// TwinCAT 3 PLC project RACBaseObjects
// Title: Base Objects Library
// Company: JABIL RAC LATAM
// Author: RAC Team
// ProjectVersion: 24.12.1
// Description: Base library for base devices and machines in RAC LATAM
// ProgramVersion: 3.1.4024.0
// libraries:
//   Tc2_MC2, * (Beckhoff Automation GmbH)
//   Tc2_Standard, * (Beckhoff Automation GmbH)
//   Tc2_System, * (Beckhoff Automation GmbH)
//   Tc3_Module, * (Beckhoff Automation GmbH)
// project tree:
//   DUTs/ ST_Nest.TcDUT, ST_RAC_EIP.TcDUT
//   GVLs/ Constants.TcGVL, GVL_Rails.TcGVL
//   / PlcTask.TcTTO
//   POUs/00_Interfaces/Device/ FB_Device.TcPOU, ST_Alarm.TcDUT
//   POUs/00_Interfaces/Machine/ FB_Machine.TcPOU
//   POUs/00_Interfaces/Stations/ EN_StationStatus.TcDUT, FB_Station.TcPOU
//   POUs/01-DevicesFB/Bimanual/ FB_Bimanual.TcPOU (not stored)
//   POUs/01-DevicesFB/BowlFeeder/ ST_BowlFeeder.TcDUT
//   POUs/01-DevicesFB/Conveyor/ FB_Conveyor.TcPOU
//   POUs/01-DevicesFB/Cylinder/ FB_Cylinder.TcPOU
//   POUs/01-DevicesFB/LightTower/ FB_LightTower.TcPOU
//   POUs/01-DevicesFB/Motor/ EN_MotionType.TcDUT, FB_Motor.TcPOU
//   POUs/01-DevicesFB/RejectCar/ FB_RejectCart.TcPOU
//   POUs/01-DevicesFB/Robot/ EN_RobotMessaging.TcDUT, FB_Robot.TcPOU, ST_RobotIO.TcDUT
//   POUs/01-DevicesFB/Scanner/ FB_Scanner.TcPOU
//   POUs/01-DevicesFB/TrayFeeder/ EN_TrayFeederMessaging.TcDUT, FB_TrayFeeder.TcPOU, ST_TrayFeederIO.TcDUT
//   POUs/01-DevicesFB/Vaccum/ FB_Vacuum.TcPOU
// real-time tasks:
//   TASK PlcTask: cycle T#10ms, priority 20, ADS port 350

CONFIGURATION RACBaseObjects
    RESOURCE PLC ON TwinCAT3
        TASK PlcTask(INTERVAL := T#10ms, PRIORITY := 20);
    END_RESOURCE
END_CONFIGURATION

// ---- DUTs/ST_Nest.TcDUT
TYPE ST_Nest :
	STRUCT
		railSerial				: STRING;
		controllerSerial		: STRING;
		batterySerial			: STRING;
		nestID					: USINT;
		conveyorPosition		: USINT;
		okToProcess				: BOOL				:= FALSE;
		failureMode				: STRING			:= 'N/A';
		endcapAssembled			: BOOL 				:= FALSE;
		controllerAssembled		: BOOL				:= FALSE;	
	END_STRUCT
END_TYPE

// ---- DUTs/ST_RAC_EIP.TcDUT
TYPE ST_RAC_EIP :
STRUCT
	byteArray 		: ARRAY [0..39] OF BYTE;
END_STRUCT
END_TYPE

// ---- POUs/00_Interfaces/Device/ST_Alarm.TcDUT
TYPE ST_Alarm :
STRUCT
	sCode							: STRING;
	bIsActive						: BOOL;
	bWrittenOnGeneralAlarm			: BOOL;
END_STRUCT
END_TYPE

// ---- POUs/00_Interfaces/Stations/EN_StationStatus.TcDUT
{attribute 'qualified_only'}
{attribute 'strict'}
{attribute 'to_string'}
TYPE EN_StationStatus :
(
	estopped			:=0,
	stopped				:=1,
	maintenance			:=2,
	initializing		:=3,
	idle				:=4,
	running				:=5
	);
END_TYPE

// ---- POUs/01-DevicesFB/BowlFeeder/ST_BowlFeeder.TcDUT
TYPE ST_BowlFeeder :
	STRUCT
		bOut_Vibrate			AT%Q*	: BOOL;
		bOut_BlowAlign			AT%Q*	: BOOL;
		bIn_NoMaterial			AT%I*	: BOOL;
		bIn_LowLevelMaterial	AT%I*	: BOOL;
		bIn_UnitInPosition		AT%I*	: BOOL;
	END_STRUCT
END_TYPE

// ---- POUs/01-DevicesFB/Motor/EN_MotionType.TcDUT
{attribute 'qualified_only'}
{attribute 'strict'}
{attribute 'to_string'}
TYPE EN_MotionType :
(
	idle 			:= 0,
	stop 			:= 1,
	home 			:= 2,
	jogPos 			:= 3,
	jogNeg 			:= 4,
	absolute 		:= 5,
	relative 		:= 6
);
END_TYPE

// ---- POUs/01-DevicesFB/Robot/EN_RobotMessaging.TcDUT
{attribute 'qualified_only'}
{attribute 'strict'}
{attribute 'to_string'}
TYPE EN_RobotMessaging :
(
	clearedCmd 					:=10000,
	ok							:=10001,
	retry						:=10002,
	skip						:=10003,
	retriesExceeded				:=10004,
	
	initStart					:=0,
	waitInitPermissive			:=10,
	turnMotorsOFF				:=20,
	waitRobotInAuto				:=30,
	resetEStop					:=40,
	PPToMain					:=50,
	turnMotorsON				:=60,
	startTaskExecuion			:=70,
	waitInitFinihsed			:=80,
	waitRetrievalPerm			:=210,
	stopTaskExecution			:=310,
	initEndMotorsOFF			:=320,
	initFinished				:=999,
	
	autoStarts					,
	waitingPickPerm				,
	pickingGood					,
	pickingNG					,
	waitingPieceStatus			,
	waitingPlacePerm			,
	placing						,
	placeFinished				,
	waitingRejectPerm			,
	rejecting					,
	rejectFinished				,
	autoCycleFinished			:=1999,
	
	manualRetrieval				,
	manualHomming				,
	manualPick					,
	manualCycPickTeach			,
	manualPlace					,
	manualCycPlaceTeach			,
	manualReject				,
	manualCycRejectTeach		
)DINT := clearedCmd;
END_TYPE

// ---- POUs/01-DevicesFB/Robot/ST_RobotIO.TcDUT
TYPE ST_RobotIO :
STRUCT
	uiin_ConnectionStatus					AT %I*		:UINT;
	eipInputs								AT %I*		:ST_RAC_EIP;
	eipOutputs								AT %Q*		:ST_RAC_EIP;
	
	diin_Sequencer		 					:DINT;
	diout_SequenceCmd						:DINT;
	rout_XCompensation						:REAL;
	rout_ZCompensation						:REAL;
	
	bin_EStop	 							:BOOL;
	bin_PPMoved	 							:BOOL;
	bin_MotorsOFF	 						:BOOL;
	bin_MotorsON	 						:BOOL;
	bin_SystemInputBusy	 					:BOOL;
	bin_RunchainOK	 						:BOOL;
	bin_AutoON	 							:BOOL;
	bin_MainTaskExecuting	 				:BOOL;
	bin_SMBBatery	 						:BOOL;
	bin_RobotNotMoving						:BOOL;
	
	bout_ResetEStop							:BOOL;
	bout_PPToMain							:BOOL;
	bout_MotorsOFF							:BOOL;
	bout_MotorsON							:BOOL;
	bout_Start								:BOOL;
	bout_Stop								:BOOL;
	
	bin_almRetCyl01							:BOOL;
	bin_almExtCyl01							:BOOL;
	bin_almBothSnsrCyl01					:BOOL;
	bin_almRetCyl02							:BOOL;
	bin_almExtCyl02							:BOOL;
	bin_almBothSnsrCyl02					:BOOL;
	bin_almRetCyl03							:BOOL;
	bin_almExtCyl03							:BOOL;
	bin_almBothSnsrCyl03					:BOOL;
END_STRUCT
END_TYPE

// ---- POUs/01-DevicesFB/TrayFeeder/EN_TrayFeederMessaging.TcDUT
{attribute 'qualified_only'}
{attribute 'strict'}
{attribute 'to_string'}
TYPE EN_TrayFeederMessaging :
(
	waitInitStart			:=0,
	initFinished			:=999,
	
	autoStart				:=1000,
	readyToScan				:=1400,
	scanning				:=1410,
	scanFinished			:=1490,
	readyToPick				:=1500,
	picking					:=1510,
	pickFinished			:=1590,
	autoProcessFinished		:=1999
)DINT := waitInitStart;
END_TYPE

// ---- POUs/01-DevicesFB/TrayFeeder/ST_TrayFeederIO.TcDUT
TYPE ST_TrayFeederIO :
STRUCT
	uiin_ConnectionStatus					AT %I*		:UINT;
	eipInputs								AT %I*		:ST_RAC_EIP;
	eipOutputs								AT %Q*		:ST_RAC_EIP;
	
	diin_StationStatus						:DINT;
	diin_Sequencer		 					:DINT;
	diout_SequenceCmd						:DINT;
	
	bin_ServosFailure						:BOOL;
	bin_initFinished						:BOOL;
	bin_AutoOn								:BOOL;
	bin_eStop								:BOOL;
	
	bout_Reset								:BOOL;
	bout_Start								:BOOL;
	bout_Stop								:BOOL;
	bout_Init_startPermissive				:BOOL;
	
	bout_readyToScan						:BOOL;
	bout_readyToPick						:BOOL;
	bin_SafetyBoxPlace_OutOfZone	 		:BOOL;
	bout_SafetyBoxPlace_Permissive 			:BOOL;
	
	bin_inScanningPosition					:BOOL;
	bout_scannninPieceIsOK					:BOOL;
	bout_scannninPieceIsNG					:BOOL;
	
	bin_delivery_trayReady					:BOOL;
	bout_delivery_trayChangeRequest			:BOOL;
END_STRUCT
END_TYPE

// ---- GVLs/Constants.TcGVL
{attribute 'qualified_only'}
VAR_GLOBAL CONSTANT
	
	Total_Nest						: USINT		:= 155;
	
	LoadPos							: USINT		:= 1;
	NestScanPos						: USINT		:= 2;
	EndcapAsmPos					: USINT		:= 3;
	ControllerScanPos				: USINT		:= 4;	
	BatteryConnectPos		 		: USINT		:= 5;
	ControllerAsmPos				: USINT		:= 6;
	DisplayScanPos		 			: USINT		:= 18;	
	BatteryDisconnectPos			: USINT		:= 20;
	TappingPos						: USINT		:= 23;
	
//	St01_LoadPos					: USINT		:= 1; // From quiles branch 
//	St01_EndcapAsmPos				: USINT		:= 3;
//	St01_ControllerAsmPos				: USINT		:= 4;
//	St01_BatteryAsmPos				: USINT		:= 5;
//	St01_UnloadPos					: USINT		:= 9;
						
END_VAR

// ---- GVLs/GVL_Rails.TcGVL
{attribute 'qualified_only'}
VAR_GLOBAL
		Nests	: ARRAY[1..Constants.Total_Nest] OF ST_Nest;
	
END_VAR

// ---- POUs/00_Interfaces/Device/FB_Device.TcPOU
FUNCTION_BLOCK  FB_Device
VAR_INPUT
	// Status of Master station
	diStationState 						: EN_StationStatus;
	
	// Device Identification Number
	sDeviceID							: STRING;
	
	// Stop executions
	bStopExecution						: BOOL;
	
	// Station Alarm Reset
	bAlarmReset							: BOOL;
END_VAR
VAR_OUTPUT
	// Display current active alarms in device, in a CVS file concatenating type string
	sAlarm								: STRING;
END_VAR
VAR RETAIN
	// Var to set timeout value in each step
	tmStepTimeout						: TIME		:=T#1S;
	
	// General timeout TON
	ton_StepTimeout						: TON;
	// Pulse ton
	ton_pulse							: TON;
END_VAR

METHOD AlarmCodesHandling : STRING
VAR_INPUT
	// Concatenated codes string
	sConcatCodes						:	STRING;
	// Code for add or delete
	sCode								:	STRING;
	// Device ID for add to alarm code
	sIDToAdd							:	STRING;
	// If alarm is active: TRUE
	bActive								:	BOOL;
END_VAR
VAR
	// Code with ID and separator added
	sProcessedCode						:	STRING;
	// Position where code was found
	iPosWhereFindCode					:	INT;
	// Length of code seeked
	iLengthOfCode						:	INT;
END_VAR
//	Add device ID, separator, seek code in concatenated codes string obtan position in the string and lentgh of seeked code
	sProcessedCode:= CONCAT(STR1:=sCode,STR2:=sIDToAdd);
	sProcessedCode:= CONCAT(STR1:=sProcessedCode,STR2:=',');
	iPosWhereFindCode:= FIND(STR1:=sConcatCodes,STR2:=sProcessedCode);
	iLengthOfCode:= LEN(STR:=sProcessedCode);

//	If code was not found add alarm is active add it to concatenated codes string
	IF (iPosWhereFindCode=0) AND (bActive) THEN
		AlarmCodesHandling:= CONCAT(STR1:=sConcatCodes,STR2:=sProcessedCode);
//	If code was found add alarm is not active delete it from concatenated codes string
	ELSIF (iPosWhereFindCode<>0) AND (NOT bActive) THEN
		AlarmCodesHandling:= DELETE(STR:=sConcatCodes,LEN:=iLengthOfCode,POS:=iPosWhereFindCode);
//	Default case return input value
	ELSE
		AlarmCodesHandling:= sConcatCodes;
	END_IF
END_METHOD

END_FUNCTION_BLOCK

// ---- POUs/00_Interfaces/Machine/FB_Machine.TcPOU
FUNCTION_BLOCK ABSTRACT FB_Machine EXTENDS FB_Device
VAR_INPUT
	// Init start permissive
	bInit_StartPermissive				: BOOL;
END_VAR
VAR_OUTPUT
	// Init finished
	bInit_Finished						: BOOL;
END_VAR
VAR RETAIN
	// Sequencer
	diActualSeqStep						: DINT;
	
	// Var to follow sequencer and evaluate timeout	
	diLastActiveStep					: DINT;
END_VAR

METHOD ABSTRACT Alarm
END_METHOD

METHOD ABSTRACT Auto
END_METHOD

METHOD ABSTRACT Init
END_METHOD

METHOD ABSTRACT IO
END_METHOD

METHOD MachineMain
//	Enable Setting Alarm Routine Execution
	THIS^.IO();

//	Machine state control

CASE diStationState OF
	EN_StationStatus.stopped,
	EN_StationStatus.estopped:			//Enables Stop Routine Execution
		THIS^.Stop();
	EN_StationStatus.initializing:		//Enables Init Routine Execution
		THIS^.Init();
	EN_StationStatus.idle:				//Enables Pause Routine
		THIS^.Pause();
	EN_StationStatus.running:			//Enables Auto Routine Execution
		THIS^.Auto();
	EN_StationStatus.maintenance:		//Enables Manual Routine Execution
		THIS^.Manual();
END_CASE

//	Enable Setting Alarm Routine Execution
	THIS^.Alarm();
END_METHOD

METHOD ABSTRACT Manual
END_METHOD

METHOD ABSTRACT Pause
END_METHOD

METHOD ABSTRACT Stop
END_METHOD

END_FUNCTION_BLOCK

// ---- POUs/00_Interfaces/Stations/FB_Station.TcPOU
FUNCTION_BLOCK FB_Station
VAR_INPUT
	// Whole Station Init finished
	bInitFinished						: BOOL;
	
	// All E-Stop buttons
	EmergencyStop 						: BOOL;
	// From safety project
	SafetyReady 						: BOOL;
	// All door sensors
	Interlock 							: BOOL;
END_VAR
VAR_OUTPUT
	// Station Actual Status 
	diStationState 						: EN_StationStatus;
	
	// Stop executions
	bStop								: BOOL;
	
	// Reset Alarms
	 bAlarmReset						: BOOL;
END_VAR
VAR
	bStopButton 			AT %I* 		: BOOL;
	bStartButton 			AT %I* 		: BOOL;
	bResetButton			AT %I* 		: BOOL;

	bStopInterface 						: BOOL;
	bPauseInterface 					: BOOL;
	bInitStartInterface					: BOOL;
	bAutoStartInterface 				: BOOL;
	bResetInterface						: BOOL;
	OpUser 								: BOOL;

	AutoModeSelector 		AT %I* 		: BOOL;
	PressureSwitch 			AT %I* 		: BOOL;
	
	// Delay for stoppping machine with button 
	ton_stopMachineDelay 				: TON;
	
	// Delay for starts machine with button
	ton_startInitStartButtonDelay 		: TON;
END_VAR

StatusControl();
Alarm();

METHOD Alarm
VAR_INPUT
END_VAR
END_METHOD

METHOD StatusControl
VAR_INPUT
END_VAR

VAR
	// Safe operation condition in any mode
	bSafeOperationCondition			: BOOL;
	
	// Condtion for any Auto operation mode
	bAutoAvailable					: BOOL;
	
	// Condition for Maintenance operation mode
	bManualAvailable				: BOOL;
END_VAR
//	Condition for operate machine safely in any mode
	bSafeOperationCondition					:=	SafetyReady AND Interlock AND PressureSwitch;

//	Condition for operation in Auto Mode
	bAutoAvailable							:=	bSafeOperationCondition AND AutoModeSelector;

//	Condition for operation in Maintenance Mode
	bManualAvailable						:=	bSafeOperationCondition AND OpUser AND (NOT AutoModeSelector);
	
//	Stopping machine with button delay
	ton_stopMachineDelay(IN:=bStopButton,PT:=T#3S);
	
//	Starting machine with button delay
	ton_startInitStartButtonDelay(IN:=bStartButton,PT:=T#2S);
	
//	For controlling reset general output
	bAlarmReset								:=	bResetButton OR bResetInterface;
 
//	For controlling stop general output
	bStop									:=	bStopButton OR bStopInterface;

//	For Stopping the machine
	CASE diStationState OF
		EN_StationStatus.initializing :		// Initializing
			IF (NOT bAutoAvailable) OR bPauseInterface OR bStopInterface OR bStopButton THEN	
				diStationState				:=EN_StationStatus.stopped;
			END_IF;
		EN_StationStatus.idle :				//	Idle
			IF (NOT bAutoAvailable) OR (NOT bInitFinished) OR bStopInterface OR ton_stopMachineDelay.Q  THEN
				diStationState				:=EN_StationStatus.stopped;
			END_IF;
		EN_StationStatus.running:			// Running
			IF (NOT bAutoAvailable) OR (NOT bInitFinished) OR bStopInterface THEN
				diStationState				:=EN_StationStatus.stopped;
			END_IF;
		EN_StationStatus.maintenance:		// Maintenance
			IF (NOT bManualAvailable) THEN
				diStationState				:=EN_StationStatus.stopped;
			END_IF;
		EN_StationStatus.eStopped:			// E Stopped
			IF NOT EmergencyStop THEN
				diStationState				:=EN_StationStatus.stopped;
			END_IF;
	END_CASE;

//	For setting machine in Initialization or Running
	IF bAutoAvailable THEN
		CASE diStationState OF
			EN_StationStatus.stopped:		//	Stopped
				IF bInitStartInterface OR ton_startInitStartButtonDelay.Q THEN
					diStationState			:=EN_StationStatus.initializing;
				END_IF;
			EN_StationStatus.idle:			//	Idle
				IF bAutoStartInterface OR ton_startInitStartButtonDelay.Q THEN
					diStationState			:=EN_StationStatus.running;
				END_IF;
		END_CASE;
	END_IF;

//	For setting machine in Idle mode
	CASE diStationState OF
		EN_StationStatus.initializing:		// Initializing
			IF 	bInitFinished THEN
				diStationState				:=EN_StationStatus.idle;
			END_IF;
		EN_StationStatus.running:			// Running
			IF bStopButton OR bPauseInterface THEN
				diStationState				:=EN_StationStatus.idle;
			END_IF;
	END_CASE;

//	For setting machine in Maintenance mode
	IF bManualAvailable AND (diStationState=EN_StationStatus.stopped) THEN
		diStationState						:=EN_StationStatus.maintenance;
	END_IF;

//	For setting machine in E Stopped mode
	IF (EmergencyStop) AND (diStationState<>EN_StationStatus.eStopped) THEN
		diStationState						:=EN_StationStatus.eStopped;
	END_IF;
END_METHOD

END_FUNCTION_BLOCK

// ---- POUs/01-DevicesFB/Conveyor/FB_Conveyor.TcPOU
FUNCTION_BLOCK FB_Conveyor EXTENDS FB_Machine
VAR_INPUT
	//All subproces in safe position
	bIn_SafeToMove					: BOOL;
	//All subprocess completed
	bIn_AllProcessComplete			: BOOL;
	//Distance between nests
	lrDistance						: LREAL;
	//If requires offset after home sequence
	lrOffsetPos						: LREAL;
	
	//Nest clamps control
	bIn_IsClamped					: BOOL;
	bIn_IsUnclamped					: BOOL;
END_VAR
VAR_OUTPUT
	//Move done, ready to receive from transfer
	bOut_ReadyToReceive				: BOOL;
	//Rail ready, in last position
	bOut_ReadyToSend				: BOOL;
	//Step complete
	bOut_MoveDone					: BOOL;
	
	bOut_ClampRequest				: BOOL;
	bOut_UnclampRequest				: BOOL;
	
	bSafetyBoxPlace_OutOfZone		: BOOL;
	
END_VAR
VAR
	Motor						: FB_Motor;
	
	//For rail track
	iCounter 					: USINT;
	tmpNest						: ST_Nest;
	
	bManualStep					: BOOL;
	bSensorLoadPos				: BOOL;
END_VAR

//	Run the standar main for any machine
SUPER^.MachineMain();

//	Motor instance
	Motor(						sDeviceID:='',
								bStopExecution:=bStopExecution,
								bAlarmReset:=bAlarmReset,
								diStationState:=diStationState,
								bInit_StartPermissive:=bInit_StartPermissive,
								MovementType:=,
								bExecute:=,
								bMovePermissive:=(bIn_SafeToMove AND TRUE),
								lrSpeed:=,
								lrPosition:=
								);

METHOD Alarm
END_METHOD

METHOD Auto
IF diActualSeqStep<1000 OR diActualSeqStep> 2000 THEN
	diActualSeqStep:= 1000;
END_IF

CASE diActualSeqStep OF
	1000:						//Reset variables
		bOut_MoveDone:= FALSE;
		bSafetyBoxPlace_OutOfZone:= FALSE;
		Motor.bExecute:= FALSE;
		diActualSeqStep:= 1010;
		
	1010: 					//Check conditions
		diActualSeqStep:= 1020;
		
	1020:					//Check for safety conditions to move
		//Absolute move, just once after homming
		IF bIn_SafeToMove   THEN
			//First move, absolute type, just if requires after home
			Motor.MovementType:= EN_MotionType.absolute;
			Motor.lrPosition:= THIS^.lrOffsetPos;
			
			motor.bExecute:= TRUE;
			IF Motor.bDone THEN
				diActualSeqStep:= 1050;
			END_IF
		END_IF
	
	1030:					//Reset variables and wait for motor done false
		Motor.bExecute:= FALSE;
		bOut_MoveDone:= FALSE;
		IF NOT Motor.bDone THEN
			diActualSeqStep:= 1040;
		END_IF
		
	1040:					//Step move	
		bOut_MoveDone:= FALSE;
		IF bIn_SafeToMove THEN
			Motor.MovementType:= EN_MotionType.relative;
			Motor.lrPosition:= lrDistance;
			
			Motor.bExecute:= TRUE;
			IF Motor.bDone THEN
				diActualSeqStep:=1050;		
			END_IF
		END_IF
		
	1050:					//Update the rail positions
		fnUpdateRailPosition();
		diActualSeqStep:= 1060;
		
	1060:					//Send the move complete
		bOut_MoveDone:= TRUE;
		IF bIn_AllProcessComplete THEN
			bOut_MoveDone:= FALSE;
			diActualSeqStep:= 1070;
		END_IF
	
	1070:					//Handshake, wait for the process complete fall
		IF NOT bIn_AllProcessComplete THEN
			diActualSeqStep:= 1080;
		END_IF
	
	1080:					//Confirm for safety conditions
		IF bIn_SafeToMove THEN
			diActualSeqStep:= 1090;
		END_IF
	1100:					//Return sequence
		diActualSeqStep:= 1030;
	
END_CASE
END_METHOD

ACTION fnUpdateRailPosition:

//Save the last nest info
tmpNest:= GVL_Rails.Nests[Constants.Total_Nest];

//Update in 1 every nest info from top to bottom
FOR iCounter:= Constants.Total_Nest - 1 TO 0 BY -1 DO
	GVL_Rails.Nests[iCounter +1] :=  GVL_Rails.Nests [iCounter];	
END_FOR

//Update the first position by the saved info
GVL_Rails.Nests[1]:= tmpNest;
END_ACTION

METHOD Init
CASE  diActualSeqStep OF
	0:					//Reset variables and stop motor
		Motor.bStopExecution:= TRUE;
		IF NOT Motor.bMotorMoving THEN
			diActualSeqStep:= 10;
		END_IF
		
	10:					//Check status
		diActualSeqStep:= 20;
		
	20:					//Wait for the initial permisive
		IF bInit_StartPermissive THEN
			diActualSeqStep:= 30;
		END_IF
		
	30: 				//Unlock cylinder
		bOut_ClampRequest:= FALSE;
		bOut_UnclampRequest:= TRUE;
		
		IF bIn_IsUnclamped THEN
			bOut_UnclampRequest:= FALSE;
			diActualSeqStep:= 40;
		END_IF
		
	40: 				//Run Motor Init to Home sequence
		Motor.Init();
		IF Motor.bInit_Finished THEN
			diActualSeqStep:= 50;	
		END_IF
				
	50:					//Initial done
		bInit_Finished:= TRUE;
		diActualSeqStep:= 1000;	
		
END_CASE
END_METHOD

METHOD IO
END_METHOD

METHOD Manual

VAR
	r_trig						: R_TRIG;
END_VAR
IF bManualStep THEN
	r_trig(clk:= TRUE);
	IF r_trig.Q THEN				//Update params only once
		Motor.MovementType:= EN_MotionType.relative;
		Motor.lrPosition:= Motor.lrActualPosition+ lrDistance;
		Motor.bExecute:= FALSE;
			
	END_IF
		Motor.bExecute:= TRUE;
	
	IF Motor.bDone THEN
		bManualStep:= FALSE;
		Motor.bExecute:= FALSE;
	END_IF	
ELSE
	
	Motor.bExecute:= FALSE;


END_IF
END_METHOD

METHOD Pause
END_METHOD

METHOD Stop
END_METHOD

END_FUNCTION_BLOCK

// ---- POUs/01-DevicesFB/Motor/FB_Motor.TcPOU
FUNCTION_BLOCK FB_Motor EXTENDS FB_Machine
VAR_INPUT
	// Movement type
	MovementType						: EN_MotionType				:=EN_MotionType.stop;
	
	// Trigger to execute configured command
	bExecute							: BOOL						:= FALSE;
	
	// Movements permissive
	bMovePermissive						: BOOL						:= FALSE;
	
	// Movement Speed
	lrSpeed								: LREAL						:= 0;
	
	// Position to reach
	lrPosition							: LREAL						:= 0;
END_VAR
VAR_OUTPUT
	bDone								: BOOL						:= FALSE;
	bMotorMoving						: BOOL						:= FALSE;
	lrActualPosition					: LREAL						:= 0;
END_VAR
VAR
	// HMI disable motor for manual manipulation
	bDisableMotor						: BOOL						:= FALSE;
	bMotorEN							: BOOL						:= FALSE;
	bMotorStop							: BOOL						:= FALSE;
	bMotorPause							: BOOL						:= FALSE;
	bMotorErrorReset					: BOOL						:= FALSE;
	bJogPos								: BOOL						:= FALSE;
	bJogNeg								: BOOL						:= FALSE;
	bTrigger							: BOOL						:= FALSE;
	bTargetPositionNoMatch				: BOOL						:= FALSE;
	lrOverride							: LREAL						:= 0;
	lrTargetPosition					: LREAL						:= 0;
	lrPositionWhenTrig					: LREAL						:= 0;
	lrActualVelocity					: LREAL						:= 0;
	lrActualAcc							: LREAL						:= 0;
	lrActualTorque						: LREAL						:= 0;
	lrActualTargetPos					: LREAL						:= 0;
	Motor								: TC2_MC2.AXIS_REF;
	mcPower								: TC2_MC2.MC_Power;
	mcMoveAbs							: TC2_MC2.MC_MoveAbsolute;
	mcMoveRel							: TC2_MC2.MC_MoveRelative;
	mcPauseMove							: TC2_MC2.MC_Halt;
	mcStopMove							: TC2_MC2.MC_Stop;
	mcJog								: TC2_MC2.MC_Jog;
	mcHomeMove							: TC2_MC2.MC_Home;
	mcReset								: TC2_MC2.MC_Reset;
END_VAR

// If station indicates stop execution reset sequence value
	IF bStopExecution THEN
		diActualSeqStep 				:= 0;
	END_IF

// Update status
	Motor.ReadStatus();

// For clearing servo errors
	mcReset(		Axis				:= Motor,
					Execute				:= ((bAlarmReset OR bMotorErrorReset) AND Motor.Status.Error));

// For enablng motor
	// If motor is not enabled, station status is different to e_stopped and DisableMotor input bit is false: Enable motor
	bMotorEN:= Motor.Status.Disabled AND (diStationState <> EN_StationStatus.estopped) AND (NOT bDisableMotor);
	mcPower(		Axis				:= Motor,
					Enable				:= bMotorEN,
					Enable_Positive		:= bMotorEN,
					Enable_Negative		:= bMotorEN,
					Override			:= lrOverride);

// Station status main
SUPER^.MachineMain();

// For auto and mintenance station status, depending on the motion type input: motor operates	
IF bMovePermissive AND ((diStationState=EN_StationStatus.running) OR (diStationState=EN_StationStatus.maintenance)) THEN
	CASE MovementType OF
		// For finding origin refference in auto and manual station state
		EN_MotionType.home:
		mcHomeMove(		Axis				:= Motor,
						Execute				:= bTrigger,
						HomingMode			:= TC2_MC2.MC_HomingMode.MC_DefaultHoming);
						
		// For jogging in auto and manual station state
		EN_MotionType.jogNeg, EN_MotionType.jogPos:
		mcJog(			Axis				:= Motor,
						JogForward			:= NOT Motor.Status.Moving AND bJogPos,
						JogBackwards		:= NOT Motor.Status.Moving AND bJogNeg,
						Mode				:= TC2_MC2.E_JogMode.MC_JOGMODE_CONTINOUS,
						Velocity			:= lrSpeed);
						
		// For executing relative movements in auto and manual station state
		EN_MotionType.relative:	
		mcMoveRel(		Axis				:= Motor,
						Execute				:= (NOT Motor.Status.Moving AND bTrigger),
						Distance			:= lrTargetPosition,
						Velocity			:= lrSpeed);
						
		// For executing absolute movements in auto and manual station state						
		EN_MotionType.absolute:
		mcMoveAbs(		Axis				:= Motor,
						Execute				:= (NOT Motor.Status.Moving AND bTrigger),
						Position			:= lrTargetPosition,
						Velocity			:= lrSpeed);
	END_CASE
	bTrigger							:= FALSE;
END_IF

// For pausing actual movement
	mcPauseMove(	Axis				:= Motor,
					Execute				:= bMotorPause AND Motor.Status.Moving);
	IF bMotorPause THEN
		bMotorPause						:= Motor.Status.Moving;
	END_IF

// For stopping actual movement
	mcStopMove(		Axis				:= Motor,
					execute				:= ((bStopExecution OR bMotorStop OR (NOT bMovePermissive)) AND Motor.Status.Moving));
	IF bMotorStop THEN
		bMotorStop						:= Motor.Status.Moving;		
	END_IF

METHOD PRIVATE Alarm
VAR
	// R Trigger VAr
	rTrigger							: R_TRIG;
	// Step in wich timeout occur
	diTimeoutStep						: DINT;
	// Actual Timed Out Sequence Step Code
	sSequenceCode						: STRING;
	
	// Async Process Concatenated Alarm Codes
	sAsyncAlarmCodes					: STRING;
END_VAR
// Timeout preset valuie setting
IF ton_StepTimeout.PT<>tmStepTimeout THEN
	ton_StepTimeout.PT					:= tmStepTimeout;
END_IF

// TON for step timeout
ton_StepTimeout(IN:=((NOT ton_StepTimeout.Q) AND (diLastActiveStep=diActualSeqStep)));

// Following of sequence for setting timeout
	IF diLastActiveStep<>diActualSeqStep THEN
		diLastActiveStep					:= diActualSeqStep;
	END_IF

// For setting acual timed out step alarm code
	rTrigger(CLK:=ton_StepTimeout.Q);
	IF rTrigger.Q THEN
		diTimeoutStep := diActualSeqStep;
		CASE diTimeoutStep OF
		// Init process timeouts
			0:										sSequenceCode := 'ISERVPRO01';
			10:										sSequenceCode := 'ESERVPRO01';
			20:										sSequenceCode := 'ESERVTIM01';
		// Auto / Manual process timeout
			1001, 2001:								sSequenceCode := 'ESERVPOS01';
			1010, 2010:								sSequenceCode := 'ESERVTIM01';
			1011, 2011:								sSequenceCode := 'ESERVTIM02';
			1012, 2012:								sSequenceCode := 'ESERVTIM02';
		END_CASE
		sSequenceCode:= CONCAT(STR1:=sSequenceCode,STR2:=sDeviceID);
		sSequenceCode:= CONCAT(STR1:=sSequenceCode,STR2:=',');
	END_IF

// For deleting last sequence alarm code automatically
	IF (diActualSeqStep<>diTimeoutStep AND diTimeoutStep<>0)THEN
		sSequenceCode:= '';
		diTimeoutStep:= 0;
	END_IF

// For setting no lineal processes alarms
	//If not homed
	sAsyncAlarmCodes:= AlarmCodesHandling(sConcatCodes:=sAsyncAlarmCodes,sCode:='SSERVPOS01',sIDToAdd:=sDeviceID,bActive:=(NOT (Motor.Status.Homed OR Motor.Status.Homing)));
	// If do not have safe move condition
	sAsyncAlarmCodes:= AlarmCodesHandling(sConcatCodes:=sAsyncAlarmCodes,sCode:='SSERVSEC01',sIDToAdd:=sDeviceID,bActive:=(NOT bMovePermissive));
	// If servo has an alarm
	sAsyncAlarmCodes:= AlarmCodesHandling(sConcatCodes:=sAsyncAlarmCodes,sCode:='ESERVALA02',sIDToAdd:=sDeviceID,bActive:=Motor.Status.Error);
	
// Concat all alarm codes
	sAlarm:= CONCAT(STR1:=sSequenceCode,STR2:=sAsyncAlarmCodes);
END_METHOD

METHOD Auto
//Update the speed if value chages
	IF Motor.PlcToNc.Override<>100 THEN
		lrOverride 						:= 100;
	END_IF

// Keep sequencer in range
	IF (diActualSeqStep<1000) OR (diActualSeqStep>1999) THEN
		diActualSeqStep					:= 1000;
	END_IF

// General sequence for executing movemen
	MovementExecution(diInitialStep:=1000);
END_METHOD

METHOD Init
VAR
	bGoHome								: BOOL;
END_VAR
//Update the speed if value chages
	IF Motor.PlcToNc.Override<>30 THEN
		lrOverride 						:= 30;
	END_IF

// Keep sequencer in range
	IF (diActualSeqStep<0) OR (diActualSeqStep>999) THEN
		diActualSeqStep					:= 0;
	END_IF

// Initialization Steps
CASE diActualSeqStep OF
	0:		// Wait Init start permissive
		tmStepTimeout					:= T#10S;	// ISERVPRO01
		bInit_Finished					:= FALSE;
		IF bInit_StartPermissive THEN
			diActualSeqStep				:=10; 
		END_IF
		
	10:		// Check if motor have error and try of reset them
		tmStepTimeout					:= T#500MS;	// ESERVPRO01
		bMotorErrorReset 				:= ((Motor.Status.Error) AND (NOT ton_StepTimeout.Q));
		IF NOT Motor.Status.Error THEN
			bMotorErrorReset			:= FALSE;
			diActualSeqStep				:= 20;
		END_IF
		
	20:		// Motor search home refference
		tmStepTimeout					:= T#50S;	// ESERVTIM01
		bGoHome							:= NOT ton_StepTimeout.Q;
		bInit_Finished					:= mcHomeMove.Done;
		IF bInit_Finished THEN
			bGoHome						:= FALSE;
			diActualSeqStep				:= 999; 
		END_IF
END_CASE

// Homming FB only for  initialization
mcHomeMove(		Axis				:= Motor,
				Execute				:= bGoHome,
				HomingMode			:= TC2_MC2.MC_HomingMode.MC_DefaultHoming);
END_METHOD

METHOD IO
bMotorMoving								:= Motor.Status.Moving;
lrActualPosition							:= Motor.NcToPlc.ActPos;
lrActualVelocity							:= Motor.NcToPlc.ActVelo;
lrActualAcc									:= Motor.NcToPlc.ActAcc;
lrActualTorque								:= Motor.NcToPlc.ActTorque;
lrActualTargetPos							:= Motor.NcToPlc.TargetPos;
END_METHOD

METHOD Manual
//Update the speed if value chages
	IF Motor.PlcToNc.Override<>30 THEN
		lrOverride := 30;
	END_IF
	
// Keep sequencer in range
	IF (diActualSeqStep<2000) OR (diActualSeqStep>2999) THEN
		diActualSeqStep					:= 2000;
	END_IF

// For jogging motor
IF MovementType = EN_MotionType.jogNeg THEN
	bJogPos:= 	FALSE;
	bJogNeg:=	 bExecute;
ELSIF MovementType = EN_MotionType.jogPos THEN
	bJogPos:= 	bExecute;
	bJogNeg:=	FALSE;
ELSE
	bJogPos:= 	FALSE;
	bJogNeg:=	FALSE;
	
	// General sequence for executing movemen
	MovementExecution(diInitialStep:=2000);
END_IF
END_METHOD

METHOD MovementExecution
VAR_INPUT
	diInitialStep						: DINT;
END_VAR
VAR
	diStartMoveStp						: DINT;
	diWaitHomeFinishedStp				: DINT;
	diWaitAbsFinishStp					: DINT;
	diWaitRelFinishStp					: DINT;
	diFinalStp							: DINT;
END_VAR
diStartMoveStp						:= diInitialStep+1;
diWaitHomeFinishedStp				:= diInitialStep+10;
diWaitAbsFinishStp					:= diInitialStep+11;
diWaitRelFinishStp					:= diInitialStep+12;
diFinalStp							:= diInitialStep+999;

// Wait start movement trigger
IF diActualSeqStep = diInitialStep THEN
	tmStepTimeout					:= T#5000S;	// No alarm
	
	// Latch when Execute input is on
	IF bExecute THEN
		lrPositionWhenTrig			:= lrActualPosition;
		lrTargetPosition			:= lrPosition;
		bTrigger					:= TRUE;
		bDone						:= FALSE;
		diActualSeqStep				:= diStartMoveStp;
	END_IF
END_IF

// Start movement
IF diActualSeqStep = diStartMoveStp THEN
	tmStepTimeout					:= T#50MS;	// ESERVPOS01
	
	CASE MovementType OF
		EN_MotionType.home :
			IF Motor.Status.HomingBusy THEN
				diActualSeqStep	:= diWaitHomeFinishedStp;
			END_IF
		EN_MotionType.absolute :
			IF Motor.Status.Moving THEN
				diActualSeqStep	:= diWaitAbsFinishStp;
			END_IF
		EN_MotionType.relative :
			lrPositionWhenTrig	:= Motor.NcToPlc.ActPos;
			lrTargetPosition	:= lrPosition;
			IF Motor.Status.Moving THEN
				diActualSeqStep	:= diWaitRelFinishStp;
			END_IF
	END_CASE
END_IF

// Wait home finished
IF diActualSeqStep = diWaitHomeFinishedStp THEN	
	tmStepTimeout					:= T#10S;	// ESERVTIM01
	IF Motor.Status.Homed THEN
		diActualSeqStep				:= diFinalStp;
	END_IF
END_IF

// Wait absolute movement finished
IF diActualSeqStep = diWaitAbsFinishStp THEN	
	tmStepTimeout					:= T#5S;	// ESERVTIM02
	IF Motor.Status.InTargetPosition THEN
		IF lrTargetPosition = Motor.NcToPlc.ActPos THEN
			bTargetPositionNoMatch	:= FALSE;
			diActualSeqStep			:=	diFinalStp;
		ELSE
			bTargetPositionNoMatch	:= TRUE;
		END_IF
	END_IF
END_IF

// Wait relative movement finished
IF diActualSeqStep = diWaitRelFinishStp THEN
	tmStepTimeout					:= T#5S;	// ESERVTIM02
	IF Motor.Status.InTargetPosition THEN
		IF (lrPositionWhenTrig + lrTargetPosition) = Motor.NcToPlc.ActPos THEN
			bTargetPositionNoMatch	:= FALSE;
			diActualSeqStep			:=	diFinalStp;
		ELSE
			bTargetPositionNoMatch	:= TRUE;
		END_IF
	END_IF
END_IF

// Auto cycle completed
IF diActualSeqStep = diFinalStp THEN	
	bDone							:= TRUE;
	diActualSeqStep					:= diInitialStep;
END_IF
END_METHOD

METHOD Pause
bMotorPause						:= Motor.Status.Moving;
END_METHOD

METHOD Stop
bInit_Finished					:= FALSE;
bMotorStop 						:= Motor.Status.Moving;
END_METHOD

END_FUNCTION_BLOCK

// ---- POUs/01-DevicesFB/Cylinder/FB_Cylinder.TcPOU
FUNCTION_BLOCK FB_Cylinder EXTENDS FB_Device
VAR_INPUT			
	bExtendRequest					: BOOL;
	bRetractRequest					: BOOL;	
	
	bPermisiveExtend				: BOOL;
	bPermisiveRetract				: BOOL;			
	
//	Time for alarm setting
	Timeout							: TIME;
END_VAR
VAR_OUTPUT
	bIsExtended						: BOOL;
	bIsRetracted					: BOOL;
END_VAR
VAR
	bAutoExecutionOK				: BOOL;
	bManualExecutionOK				: BOOL;
	bIsExtending					: BOOL;
	bIsRetracting					: BOOL;
	bExecuteExtend					: BOOL;
	bExecuteRetract					: BOOL;

//	Cylinder extend output
	bValveExtend					AT %Q* : BOOL;
//	Cylinder retract output
	bValveRetract 					AT %Q* : BOOL;
	
//	Clinder extended sensor
	bSensorExtended					AT %I* : BOOL;
//	Clinder retracted sensor
	bSensorRetracted				AT %I* : BOOL;
END_VAR

//	Conditions to move cylinder
	bAutoExecutionOK		:= (diStationState=EN_StationStatus.running) AND (NOT bStopExecution);
	bManualExecutionOK		:= (diStationState=EN_StationStatus.maintenance) AND (NOT bStopExecution);
	bExecuteExtend			:= ((bAutoExecutionOK OR bManualExecutionOK) AND bPermisiveExtend AND bExtendRequest AND (NOT bRetractRequest));
	bExecuteRetract			:= ((bAutoExecutionOK OR bManualExecutionOK) AND bPermisiveRetract AND (NOT bExtendRequest) AND bRetractRequest);

// If conditions for moving then move cylinder
	IF bExecuteExtend OR bExecuteRetract THEN 
		//	Extend cylinder valve
			bValveExtend	:= bExecuteExtend;
		//	Retract cylinder valve
			bValveRetract	:= bExecuteRetract;
	END_IF

//	Conditions for considerate is executing and no reaching position
	bIsExtending			:= bValveExtend AND (NOT bSensorExtended);
	bIsRetracting			:= bValveRetract AND (NOT bSensorRetracted);
//	Assign value to function block status
	bIsExtended				:= bSensorExtended AND NOT bSensorRetracted;
	bIsRetracted			:= bSensorRetracted AND NOT bSensorExtended;

//	For setting alarms
	Alarm();

METHOD Alarm
VAR 
	bAlm_ExtendReqWithoutPerm		: BOOL;
	bAlm_RetractReqWithoutPerm		: BOOL;
	bAlm_BohSensors					: BOOL;
	bAlm_BothActions				: BOOL;
	bAlm_ReqActionNoValidOper		: BOOL;
END_VAR
//	Timer for set action executing timeout alarm
	ton_StepTimeout(		IN:=bIsExtending OR bIsRetracting,
							PT:=Timeout);

//	Extending request without permissive
	IF bExtendRequest AND (NOT bPermisiveExtend) THEN
		bAlm_ExtendReqWithoutPerm		:=TRUE;
	END_IF

//	Retracting request without permissive
	IF bRetractRequest AND (NOT bPermisiveRetract) THEN
		bAlm_RetractReqWithoutPerm		:=TRUE;
	END_IF

//	Both sensors active
	IF bSensorExtended AND bSensorRetracted THEN
		bAlm_BohSensors					:=TRUE;
	END_IF

//	Both actions requested
	IF bRetractRequest AND (NOT bPermisiveRetract) THEN
		bAlm_BothActions				:=TRUE;
	END_IF

//	Action request with no valid operation mode
	IF (bExtendRequest OR bRetractRequest) AND (NOT bAutoExecutionOK) AND (NOT bManualExecutionOK) THEN
		bAlm_ReqActionNoValidOper		:=TRUE;
	END_IF

//	General alarm reset
	IF bAlarmReset THEN
		bAlm_ExtendReqWithoutPerm		:= FALSE;
		bAlm_RetractReqWithoutPerm		:= FALSE;
		bAlm_BohSensors					:= FALSE;
		bAlm_BothActions				:= FALSE;
		bAlm_ReqActionNoValidOper		:= FALSE;
	END_IF

//	For extension timeout alarm setting
	AlarmCodesHandling(sConcatCodes:=sAlarm,sCode:='WCYLISTU01',sIDToAdd:=sDeviceID,bActive:=(bIsExtending AND ton_StepTimeout.Q));
//	For retraction timeout alarm setting
	AlarmCodesHandling(sConcatCodes:=sAlarm,sCode:='WCYLISTU02',sIDToAdd:=sDeviceID,bActive:=(bIsRetracting AND ton_StepTimeout.Q));
//	For extension request without permissive alarm setting
	AlarmCodesHandling(sConcatCodes:=sAlarm,sCode:='WCYLIGEN01',sIDToAdd:=sDeviceID,bActive:=bAlm_ExtendReqWithoutPerm);
//	For retraction request without permissive alarm setting
	AlarmCodesHandling(sConcatCodes:=sAlarm,sCode:='WCYLIGEN02',sIDToAdd:=sDeviceID,bActive:=bAlm_RetractReqWithoutPerm);
//	For both sensors detected alarm setting
	AlarmCodesHandling(sConcatCodes:=sAlarm,sCode:='WCYLIDET01',sIDToAdd:=sDeviceID,bActive:=bAlm_BohSensors);
//	For both actions requested simultaneously alarm setting
	AlarmCodesHandling(sConcatCodes:=sAlarm,sCode:='ECYLIOMD01',sIDToAdd:=sDeviceID,bActive:=bAlm_BothActions);
//	For request action in no valid operation mode alarm setting
	AlarmCodesHandling(sConcatCodes:=sAlarm,sCode:='ECYLIOMD02',sIDToAdd:=sDeviceID,bActive:=bAlm_ReqActionNoValidOper);
END_METHOD

END_FUNCTION_BLOCK

// ---- POUs/01-DevicesFB/LightTower/FB_LightTower.TcPOU
FUNCTION_BLOCK FB_LightTower EXTENDS FB_Device
VAR_INPUT
	diStationState					: EN_StationStatus;
END_VAR
VAR
	Green	 			AT %Q* 		:BOOL;
	Ambar	 			AT %Q* 		:BOOL;
	Red		 			AT %Q* 		:BOOL;
	Buzzer 				AT %Q* 		:BOOL;
END_VAR

END_FUNCTION_BLOCK

// ---- POUs/01-DevicesFB/RejectCar/FB_RejectCart.TcPOU
FUNCTION_BLOCK FB_RejectCart EXTENDS FB_Machine
VAR_INPUT
	// Device identification
	sLockCylinerID					: STRING;
	
	// Safety box permissive for release and remove cart
	bSafetyBox_permissive			: BOOL;
	
	// Reject request
	bPlacePieceOnCartRequest		: BOOL;
END_VAR
VAR_OUTPUT
	// Safety box enter permissive
	bSafetyBox_okForEnter			: BOOL;
	
	// Request for pieces removal when cart is full
	bRemovePiecesRequest			: BOOL;
	
	// Sensors presence array
	byAvailableNests				: ARRAY[0..7] OF BOOL;
END_VAR
VAR
	// Timmers for considering cart in place
	tonCartIsInPlace				: TON;
	
	// Timmers for considering cart removed
	tonCartRemoved					: TON;

	// Occuped nests in reject cart
	siOccupedNests					: SINT;
	
	// Cart is in position sensor
	bCartPresence					AT %I* : BOOL;
	// 8 sensor array
	byRejectNestsSensors			AT %I* : ARRAY[0..7] OF BOOL;

	// Cylinder for locking the cart in place
	fbCartLock						: FB_Cylinder;
END_VAR

	CountNests();

//	Run the standar main for any machine
	SUPER^.MachineMain();

//	Safety permisive conditions for any device
	fbCartLock(						diStationState:=diStationState,
									sDeviceID:='',
									bStopExecution:=bStopExecution,
									bAlarmReset:=bAlarmReset,
									bPermisiveExtend:= bCartPresence AND bSafetyBox_permissive,
									bPermisiveRetract:= bCartPresence AND bSafetyBox_permissive,
									Timeout:= T#1S);
	fbCartLock.bExtendRequest		:=FALSE;
	fbCartLock.bRetractRequest		:=FALSE;

METHOD  Alarm
//	Step timeout
	ton_StepTimeout(					IN:= diActualSeqStep=diLastActiveStep,
										PT:= T#1S);

// 	Following of sequence for setting timeout
	IF diLastActiveStep<>diActualSeqStep THEN
		diLastActiveStep					:= diActualSeqStep;
	END_IF

//	For setting an sequence alarm code
	IF ton_StepTimeout.Q THEN
		CASE diActualSeqStep OF
			10: 	sAlarm				:= '';	// Init wait cart in position timeout
			50: 	sAlarm				:= '';	// Cart clamping timeout
			110: 	sAlarm				:= '';	// Cart removal timeout
			1000: 	sAlarm				:= '';	// Cart in position and clamped timeout
			1100: 	sAlarm				:= '';	// Cart removal timeout
		END_CASE
	END_IF

//	Concat general alarm codes with cart lock cylinder alarm codes
	sAlarm								:= CONCAT(STR1:=sAlarm,STR2:=fbCartLock.sAlarm);
END_METHOD

METHOD  Auto
//	Keep sequencer in range
	IF diActualSeqStep<1000 OR diActualSeqStep>1999 THEN
		diActualSeqStep					:= 1000;
	END_IF

CASE diActualSeqStep OF
	1000:								//	Check for cart in position and it is clamped
		IF tonCartIsInPlace.Q AND fbCartLock.bIsExtended THEN
			fbCartLock.bRetractRequest	:= FALSE;
			fbCartLock.bExtendRequest	:= FALSE;
			diActualSeqStep				:= 1050;
	
		ELSIF tonCartIsInPlace.Q AND fbCartLock.bIsRetracted THEN
			fbCartLock.bRetractRequest	:= FALSE;
			fbCartLock.bExtendRequest	:= TRUE;
	
		ELSE
			fbCartLock.bExtendRequest	:= FALSE;
			fbCartLock.bRetractRequest	:= TRUE;
		END_IF
	1050:								//	If there are not availability of places in cart release it and wait it has been removed
		IF siOccupedNests>=8 THEN
			fbCartLock.bExtendRequest	:= FALSE;
			fbCartLock.bRetractRequest	:= TRUE;
		END_IF
		IF fbCartLock.bIsRetracted THEN
			diActualSeqStep				:= 1100;
		END_IF
	1100:								//	Waiting cart removal
		IF tonCartRemoved.Q THEN
			diActualSeqStep				:= 1000;
		END_IF
END_CASE
END_METHOD

METHOD CountNests
VAR
	indexCountOccuped					: INT;
END_VAR
//  Counts occuped nests in the cart
	siOccupedNests					:= 0;
	FOR indexCountOccuped:=0 TO 7 BY 1 DO
		IF byRejectNestsSensors[indexCountOccuped] THEN
			siOccupedNests				:= siOccupedNests + 1;
		END_IF
	END_FOR;
END_METHOD

METHOD  Init
//	Keep sequencer in range
	IF diActualSeqStep<0 OR diActualSeqStep>999 THEN
		diActualSeqStep					:= 0;
	END_IF

CASE diActualSeqStep OF
	0:									//	Wait for the initial permisive and reset values
		IF  bInit_StartPermissive THEN
			fbCartLock.bRetractRequest	:= FALSE;
			fbCartLock.bExtendRequest	:= FALSE;
			diActualSeqStep 			:= 10;
		END_IF
	10:									// Check cart is in place
		IF tonCartIsInPlace.Q THEN
			diActualSeqStep 			:= 50;
		ELSE
			fbCartLock.bRetractRequest:=TRUE;
		END_IF
	50:									// Confirm cart is clamped
		fbCartLock.bRetractRequest		:= FALSE;
		fbCartLock.bExtendRequest		:= TRUE;
		IF fbCartLock.bIsExtended THEN
			fbCartLock.bExtendRequest	:= FALSE;
			diActualSeqStep				:= 110;
		END_IF
	110:								// Check reject nest availability for release cart
		IF siOccupedNests>=4 THEN
			diActualSeqStep				:= 150;
		ELSE
			diActualSeqStep 			:= 999;
		END_IF
	150:								// Unlock cart and wait it's removed
		bRemovePiecesRequest			:= TRUE;
		fbCartLock.bRetractRequest		:= TRUE;
		IF fbCartLock.bIsRetracted AND tonCartRemoved.Q THEN
			diActualSeqStep				:= 0;
		END_IF
	999:								// Init finished
		bInit_Finished					:= TRUE;
END_CASE
END_METHOD

METHOD  IO
VAR
	indexIO									: INT;
END_VAR
//	For considering cart in place
	tonCartIsInPlace(						IN:=bCartPresence,
											PT:=T#1S);

//	For considering cart has been removed
	tonCartRemoved(							IN:=NOT bCartPresence,
												PT:=T#1S);

//	If all places are ocupped request cart removal
	IF siOccupedNests>=8 THEN
		bRemovePiecesRequest				:= TRUE;
//	If cart is removed clear request
	ELSIF tonCartRemoved.Q THEN
		bRemovePiecesRequest				:= FALSE;
	END_IF

//	Piece sensor inverse polaritiy refreshing in available positions var
	IF tonCartIsInPlace.Q AND fbCartLock.bIsExtended THEN
		FOR indexIO:=0 TO 7 BY 1 DO
			byAvailableNests[indexIO]		:= NOT byRejectNestsSensors[indexIO];
		END_FOR;
	ELSE
		FOR indexIO:=0 TO 7 BY 1 DO
			byAvailableNests[indexIO]		:= FALSE;
		END_FOR;
	END_IF

//	For safety box enter permissive
	bSafetyBox_okForEnter					:= tonCartIsInPlace.Q AND fbCartLock.bIsExtended;
END_METHOD

METHOD  Manual
END_METHOD

METHOD  Pause
END_METHOD

METHOD  Stop
END_METHOD

END_FUNCTION_BLOCK

// ---- POUs/01-DevicesFB/Robot/FB_Robot.TcPOU
FUNCTION_BLOCK FB_Robot EXTENDS FB_Machine
VAR_INPUT
	// Robot move in pick zone permissive
	bSafetyBoxPick_Permissive			: BOOL;
	// Robot move in place zone permissive
	bSafetyBoxPlace_Permissive			: BOOL;
	// Robot move in pick zone permissive
	bSafetyBoxReject_Permissive			: BOOL;
	
	// Good material is on work position
	bOKMaterialReadyToPick				: BOOL;
	// NG material is on work position
	bNGMaterialReadyToPick				: BOOL;
	
	// Piece is good for process
	bPiceIsGood							: BOOL;
	// Piece is no good for process
	bPiceIsNG							: BOOL;
	
	// Material requested
	bPlace_MaterialRequest				: BOOL;
	
	// Reject material request
	bReject_MaterialRequest				: ARRAY[0..7] OF BOOL;
END_VAR
VAR_OUTPUT	
	// Robot is out of pick safety zone
	bSafetyBoxPick_OutOfZone 			: BOOL;
	// Robot is out of place safety zone
	bSafetyBoxPlace_OutOfZone 			: BOOL;
	// Robot is out of reject safety zone
	bSafetyBoxReject_OutOfZone 			: BOOL;
	
	// Ask for replace material tray
	bPick_AllMaterialPicked 			: BOOL;
	
	// Material placed
	bPlace_Done							: BOOL;
	
	// Material rejected
	bReject_Done						: BOOL;
END_VAR
VAR
	// Structure for IO Mapping
	RobotIO								: ST_RobotIO;
END_VAR
VAR RETAIN
	// Input: HMI setting for dry cycle
	bDryCycleON							: BOOL;
	// Input: HMI Permissive to init with manually jogged robot
	bRetrievalPermissive				: BOOL;
	// Input: HMI Permissive to retry pick when retries exceeded
	bPickRetryPermissive				: BOOL;
END_VAR

//	Enable Setting Alarm Routine Execution
	THIS^.IO();

//	Machine state control

CASE diStationState OF
	EN_StationStatus.stopped,
	EN_StationStatus.estopped:			//Enables Stop Routine Execution
		THIS^.Stop();
	EN_StationStatus.initializing:		//Enables Init Routine Execution
		THIS^.Init();
	EN_StationStatus.idle:				//Enables Pause Routine
		THIS^.Pause();
	EN_StationStatus.running:			//Enables Auto Routine Execution
		THIS^.Auto();
	EN_StationStatus.maintenance:		//Enables Manual Routine Execution
		THIS^.Manual();
END_CASE

//	Enable Setting Alarm Routine Execution
	THIS^.Alarm();

METHOD Alarm
VAR
	// R Trigger VAr
	rTrigger							: R_TRIG;
	// Step in wich timeout occur
	diTimeoutStep						: DINT;
	// Actual Timed Out Sequence Step Code
	sSequenceCode						: STRING;
	
	// Async Process Concatenated Alarm Codes
	sAsyncAlarmCodes					: STRING;
END_VAR
//	Compare and asign time value to timeout
	IF tmStepTimeout<>ton_StepTimeout.PT THEN
		ton_StepTimeout.PT					:=	tmStepTimeout;
	END_IF

//	General timer step timeout
	ton_StepTimeout(PT:=T#1S);
//	Pulse ton
	ton_pulse(PT:=T#100ms);

// For setting acual timed out step alarm code
	rTrigger(CLK:=ton_StepTimeout.Q);
	IF rTrigger.Q THEN
		diTimeoutStep := diActualSeqStep;
		CASE diTimeoutStep OF
		// Init process timeouts
			EN_RobotMessaging.initStart: 			sSequenceCode := 'EROBOPRO02';
			EN_RobotMessaging.turnMotorsOFF: 		sSequenceCode := 'WROBOPRO04';
			EN_RobotMessaging.resetEStop:			sSequenceCode := 'SROBOSEC01';
			EN_RobotMessaging.PPToMain:				sSequenceCode := 'EROBOPRO04';
			EN_RobotMessaging.turnMotorsON:			sSequenceCode := 'WROBOPRO03';
			EN_RobotMessaging.startTaskExecuion:	sSequenceCode := 'EROBOPRO03';
			EN_RobotMessaging.waitInitFinihsed:		sSequenceCode := 'WROBOPRO02';
			EN_RobotMessaging.waitRetrievalPerm:	sSequenceCode := 'EROBOPOS01';
			EN_RobotMessaging.stopTaskExecution:	sSequenceCode := 'EROBOPRO02';
			
		// Robot Auto
			EN_RobotMessaging.autoStarts:			sSequenceCode := 'IROBOTIM01';
			EN_RobotMessaging.waitingPickPerm:		sSequenceCode := 'IROBOTIM02';
			EN_RobotMessaging.pickingGood,
			EN_RobotMessaging.pickingNG:			sSequenceCode := 'IROBOTIM03';
			EN_RobotMessaging.waitingPieceStatus:	sSequenceCode := 'IROBOTIM04';
			EN_RobotMessaging.waitingPlacePerm:		sSequenceCode := 'IROBOTIM05';
			EN_RobotMessaging.placing:				sSequenceCode := 'IROBOTIM06';
			EN_RobotMessaging.placeFinished:		sSequenceCode := 'IROBOTIM07';
			EN_RobotMessaging.waitingRejectPerm:	sSequenceCode := 'IROBOTIM08';
			EN_RobotMessaging.rejecting:			sSequenceCode := 'IROBOTIM09';
			EN_RobotMessaging.rejectFinished:		sSequenceCode := 'IROBOTIM10';
		END_CASE
		sSequenceCode:= CONCAT(STR1:=sSequenceCode,STR2:=sDeviceID);
		sSequenceCode:= CONCAT(STR1:=sSequenceCode,STR2:=',');
	END_IF

// For deleting last sequence alarm code automatically
	IF (diActualSeqStep<>diTimeoutStep AND diTimeoutStep<>EN_RobotMessaging.clearedCmd)THEN
		sSequenceCode:= '';
		diTimeoutStep:= EN_RobotMessaging.clearedCmd;
	END_IF

// For setting no lineal processes alarms
	// Robot is not in auto mode
	sAsyncAlarmCodes:= AlarmCodesHandling(sConcatCodes:=sAsyncAlarmCodes,sCode:='WROBOPRO01',sIDToAdd:=sDeviceID,bActive:=(NOT RobotIO.bin_AutoON));
	// Robot connection failed
	sAsyncAlarmCodes:= AlarmCodesHandling(sConcatCodes:=sAsyncAlarmCodes,sCode:='EROBOCON04',sIDToAdd:=sDeviceID,bActive:=(RobotIO.uiin_ConnectionStatus=0));
	// Robot Battery low
	sAsyncAlarmCodes:= AlarmCodesHandling(sConcatCodes:=sAsyncAlarmCodes,sCode:='WROBOALA01',sIDToAdd:=sDeviceID,bActive:=(NOT RobotIO.bin_SMBBatery));
	// Robot EStop pressed
	sAsyncAlarmCodes:= AlarmCodesHandling(sConcatCodes:=sAsyncAlarmCodes,sCode:='SROBOSEC01',sIDToAdd:=sDeviceID,bActive:=(NOT RobotIO.bin_EStop));
	// Robot Stucked in pick safe box
	sAsyncAlarmCodes:= AlarmCodesHandling(sConcatCodes:=sAsyncAlarmCodes,sCode:='WROBOSTU01',sIDToAdd:=sDeviceID,bActive:=((NOT bSafetyBoxPick_OutOfZone) AND (bSafetyBoxPick_Permissive)));
	// Robot Stucked in place safe box
	sAsyncAlarmCodes:= AlarmCodesHandling(sConcatCodes:=sAsyncAlarmCodes,sCode:='WROBOSTU01',sIDToAdd:=sDeviceID,bActive:=((NOT bSafetyBoxPlace_OutOfZone) AND (bSafetyBoxPlace_Permissive)));
	// Robot Stucked in reject safe box
	sAsyncAlarmCodes:= AlarmCodesHandling(sConcatCodes:=sAsyncAlarmCodes,sCode:='WROBOSTU01',sIDToAdd:=sDeviceID,bActive:=((NOT bSafetyBoxReject_OutOfZone) AND (bSafetyBoxReject_Permissive)));
	// Cylinder doesn't reach start of stroke
	sAsyncAlarmCodes:= AlarmCodesHandling(sConcatCodes:=sAsyncAlarmCodes,sCode:='WCYLISTU0201',sIDToAdd:=sDeviceID,bActive:=(RobotIO.bin_almRetCyl01));
	// Cylinder doesn't reach end of stroke
	sAsyncAlarmCodes:= AlarmCodesHandling(sConcatCodes:=sAsyncAlarmCodes,sCode:='WCYLISTU0101',sIDToAdd:=sDeviceID,bActive:=(RobotIO.bin_almExtCyl01));
	// Cylinder both sensors detected
	sAsyncAlarmCodes:= AlarmCodesHandling(sConcatCodes:=sAsyncAlarmCodes,sCode:='WCYLIDET0101',sIDToAdd:=sDeviceID,bActive:=(RobotIO.bin_almBothSnsrCyl01));
	// Cylinder doesn't reach start of stroke
	sAsyncAlarmCodes:= AlarmCodesHandling(sConcatCodes:=sAsyncAlarmCodes,sCode:='WCYLISTU0202',sIDToAdd:=sDeviceID,bActive:=(RobotIO.bin_almRetCyl02));
	// Cylinder doesn't reach end of stroke
	sAsyncAlarmCodes:= AlarmCodesHandling(sConcatCodes:=sAsyncAlarmCodes,sCode:='WCYLISTU0102',sIDToAdd:=sDeviceID,bActive:=(RobotIO.bin_almExtCyl02));
	// Cylinder both sensors detected
	sAsyncAlarmCodes:= AlarmCodesHandling(sConcatCodes:=sAsyncAlarmCodes,sCode:='WCYLIDET0102',sIDToAdd:=sDeviceID,bActive:=(RobotIO.bin_almBothSnsrCyl02));
	// Cylinder doesn't reach start of stroke
	sAsyncAlarmCodes:= AlarmCodesHandling(sConcatCodes:=sAsyncAlarmCodes,sCode:='WCYLISTU0203',sIDToAdd:=sDeviceID,bActive:=(RobotIO.bin_almRetCyl03));
	// Cylinder doesn't reach end of stroke
	sAsyncAlarmCodes:= AlarmCodesHandling(sConcatCodes:=sAsyncAlarmCodes,sCode:='WCYLISTU0103',sIDToAdd:=sDeviceID,bActive:=(RobotIO.bin_almExtCyl03));
	// Cylinder both sensors detected
	sAsyncAlarmCodes:= AlarmCodesHandling(sConcatCodes:=sAsyncAlarmCodes,sCode:='WCYLIDET0103',sIDToAdd:=sDeviceID,bActive:=(RobotIO.bin_almBothSnsrCyl03));

// Concat all alarm codes
	sAlarm:= CONCAT(STR1:=sSequenceCode,STR2:=sAsyncAlarmCodes);
END_METHOD

METHOD Auto
VAR
	indexRejectSpaces						: INT;
END_VAR
//	Keep sequencer in range
	IF (diActualSeqStep<1000) OR  (diActualSeqStep>1999) THEN 
		diActualSeqStep					:=	0;
	END_IF

CASE diActualSeqStep OF
	EN_RobotMessaging.autoStarts:			//	Motors ON and Start Auto
		ton_StepTimeout.IN					:=	RobotIO.bout_MotorsON OR RobotIO.bout_Start;
		IF tmStepTimeout<>T#1S THEN
			tmStepTimeout					:=	T#1S;
		END_IF
		
		RobotIO.bout_MotorsON				:=	RobotIO.bin_MotorsOFF AND (NOT RobotIO.bin_MotorsON);
		RobotIO.bout_Start					:=	(NOT RobotIO.bin_MainTaskExecuting) AND RobotIO.bin_MotorsON;
		
		IF RobotIO.bin_MotorsON AND (NOT RobotIO.bin_MotorsOFF) AND RobotIO.bin_MainTaskExecuting
			AND ((RobotIO.diin_Sequencer=EN_RobotMessaging.waitingPickPerm) OR (RobotIO.diin_Sequencer=EN_RobotMessaging.waitingPieceStatus)
			OR (RobotIO.diin_Sequencer=EN_RobotMessaging.waitingPlacePerm) OR (RobotIO.diin_Sequencer=EN_RobotMessaging.waitingRejectPerm)) THEN 
			ton_StepTimeout.IN				:=	FALSE;
			RobotIO.diout_SequenceCmd		:=	EN_RobotMessaging.clearedCmd;
			diActualSeqStep					:=	RobotIO.diin_Sequencer;
		END_IF
		
	EN_RobotMessaging.waitingPickPerm:		//	Robot wating for picking permiissve
		IF NOT ton_StepTimeout.Q THEN 
			ton_StepTimeout.IN				:=	TRUE;
		END_IF
		IF tmStepTimeout<>T#1S THEN
			tmStepTimeout					:=	T#1S;
		END_IF
		
		IF bOKMaterialReadyToPick AND (NOT bNGMaterialReadyToPick) THEN
			RobotIO.diout_SequenceCmd		:=	EN_RobotMessaging.pickingGood;
		ELSIF (NOT bOKMaterialReadyToPick) AND bNGMaterialReadyToPick THEN
			RobotIO.diout_SequenceCmd		:=	EN_RobotMessaging.pickingNG;
		END_IF
		
		IF (RobotIO.diin_Sequencer=RobotIO.diout_SequenceCmd) AND ((RobotIO.diout_SequenceCmd=EN_RobotMessaging.pickingGood) OR (RobotIO.diout_SequenceCmd=EN_RobotMessaging.pickingNG)) THEN 
			ton_StepTimeout.IN				:=	FALSE;
			RobotIO.diout_SequenceCmd		:=	EN_RobotMessaging.clearedCmd;
			diActualSeqStep					:=	RobotIO.diin_Sequencer;
		END_IF
		
	EN_RobotMessaging.pickingGood,
	EN_RobotMessaging.pickingNG:			//	Robot picking
		IF NOT ton_StepTimeout.Q THEN 
			ton_StepTimeout.IN				:=	TRUE;
		END_IF
		IF tmStepTimeout<>T#2S THEN
			tmStepTimeout					:=	T#2S;
		END_IF
		
		IF (RobotIO.diin_Sequencer=EN_RobotMessaging.retriesExceeded) AND bPickRetryPermissive THEN 
			RobotIO.diout_SequenceCmd		:=	en_RobotMessaging.retry;
		END_IF
		
		IF (RobotIO.diin_Sequencer=EN_RobotMessaging.waitingPieceStatus) THEN 
			ton_StepTimeout.IN				:=	FALSE;
			RobotIO.diout_SequenceCmd		:=	en_RobotMessaging.clearedCmd;
			diActualSeqStep					:=	RobotIO.diin_Sequencer;
		END_IF
		
	EN_RobotMessaging.waitingPieceStatus:	//	Waiting piece on robot status
		IF NOT ton_StepTimeout.Q THEN 
			ton_StepTimeout.IN				:=	TRUE;
		END_IF
		IF tmStepTimeout<>T#1S THEN
			tmStepTimeout					:=	T#1S;
		END_IF
		
		IF bPiceIsGood AND (NOT bPiceIsNG) THEN 
			RobotIO.diout_SequenceCmd		:=	en_RobotMessaging.waitingPlacePerm;
		ELSIF (NOT bPiceIsGood) AND bPiceIsNG THEN 
			RobotIO.diout_SequenceCmd		:=	en_RobotMessaging.waitingRejectPerm;
		END_IF
		
		IF (RobotIO.diin_Sequencer=EN_RobotMessaging.waitingPlacePerm) OR (RobotIO.diin_Sequencer=EN_RobotMessaging.waitingRejectPerm) THEN 
			ton_StepTimeout.IN				:=	FALSE;
			RobotIO.diout_SequenceCmd		:=	en_RobotMessaging.clearedCmd;
			diActualSeqStep					:=	RobotIO.diin_Sequencer;
		END_IF
		
	EN_RobotMessaging.waitingPlacePerm:		//	Wait Place Material Request
		IF NOT ton_StepTimeout.Q THEN 
			ton_StepTimeout.IN				:=	TRUE;
		END_IF
		IF tmStepTimeout<>T#2S THEN
			tmStepTimeout					:=	T#2S;
		END_IF
		
		IF bPlace_MaterialRequest THEN
			RobotIO.diout_SequenceCmd		:=	EN_RobotMessaging.placing;
		END_IF
		
		IF (RobotIO.diin_Sequencer=EN_RobotMessaging.placing) THEN 
			ton_StepTimeout.IN				:=	FALSE;
			RobotIO.diout_SequenceCmd		:=	en_RobotMessaging.clearedCmd;
			diActualSeqStep					:=	RobotIO.diin_Sequencer;
		END_IF
		
	EN_RobotMessaging.placing:				//	Placing
		IF NOT ton_StepTimeout.Q THEN 
			ton_StepTimeout.IN				:=	TRUE;
		END_IF
		IF tmStepTimeout<>T#2S THEN
			tmStepTimeout					:=	T#2S;
		END_IF
		
		IF (RobotIO.diin_Sequencer=EN_RobotMessaging.placeFinished) THEN 
			ton_StepTimeout.IN				:=	FALSE;
			RobotIO.diout_SequenceCmd		:=	en_RobotMessaging.clearedCmd;
			diActualSeqStep					:=	RobotIO.diin_Sequencer;
		END_IF
		
	EN_RobotMessaging.placeFinished:		//	Placing finished informing
		IF NOT ton_StepTimeout.Q THEN 
			ton_StepTimeout.IN				:=	TRUE;
		END_IF
		IF tmStepTimeout<>T#1S THEN
			tmStepTimeout					:=	T#1S;
		END_IF
		
		bPlace_Done							:=	TRUE;
		
		IF (NOT bPlace_MaterialRequest) THEN 
			RobotIO.diout_SequenceCmd		:=	EN_RobotMessaging.placeFinished;
		END_IF
		
		
		IF (RobotIO.diin_Sequencer<>EN_RobotMessaging.placeFinished) THEN 
			ton_StepTimeout.IN				:=	FALSE;
			RobotIO.diout_SequenceCmd		:=	en_RobotMessaging.clearedCmd;
			diActualSeqStep					:=	EN_RobotMessaging.autoCycleFinished;
		END_IF
		
	EN_RobotMessaging.waitingRejectPerm:	//	Wait reject material request
		IF NOT ton_StepTimeout.Q THEN 
			ton_StepTimeout.IN				:=	TRUE;
		END_IF
		IF tmStepTimeout<>T#2S THEN
			tmStepTimeout					:=	T#2S;
		END_IF
		
		FOR indexRejectSpaces:=0 TO 7 BY 1 DO
			IF bReject_MaterialRequest[indexRejectSpaces] THEN
				RobotIO.diout_SequenceCmd		:=	EN_RobotMessaging.rejecting;
			END_IF
		END_FOR;
		
		IF (RobotIO.diin_Sequencer=EN_RobotMessaging.rejecting) THEN 
			ton_StepTimeout.IN				:=	FALSE;
			RobotIO.diout_SequenceCmd		:=	en_RobotMessaging.clearedCmd;
			diActualSeqStep					:=	RobotIO.diin_Sequencer;
		END_IF
		
	EN_RobotMessaging.rejecting:			//	Rejecting
		IF NOT ton_StepTimeout.Q THEN 
			ton_StepTimeout.IN				:=	TRUE;
		END_IF
		IF tmStepTimeout<>T#2S THEN
			tmStepTimeout					:=	T#2S;
		END_IF
		
		IF (RobotIO.diin_Sequencer=EN_RobotMessaging.rejectFinished) THEN 
			ton_StepTimeout.IN						:=	FALSE;
			RobotIO.diout_SequenceCmd		:=	en_RobotMessaging.clearedCmd;
			diActualSeqStep					:=	RobotIO.diin_Sequencer;
		END_IF
		
	EN_RobotMessaging.rejectFinished:		//	Rejecting finished informing
		IF NOT ton_StepTimeout.Q THEN 
			ton_StepTimeout.IN				:=	TRUE;
		END_IF
		IF tmStepTimeout<>T#1S THEN
			tmStepTimeout					:=	T#1S;
		END_IF
		
		bReject_Done						:=	TRUE;
		
		FOR indexRejectSpaces:=0 TO 7 BY 1 DO
			IF bReject_MaterialRequest[indexRejectSpaces] THEN
				RobotIO.diout_SequenceCmd		:=	EN_RobotMessaging.rejectFinished;
			END_IF
		END_FOR;
		
		IF (RobotIO.diin_Sequencer<>EN_RobotMessaging.rejectFinished) THEN 
			ton_StepTimeout.IN				:=	FALSE;
			RobotIO.diout_SequenceCmd		:=	en_RobotMessaging.clearedCmd;
			diActualSeqStep					:=	EN_RobotMessaging.autoCycleFinished;
		END_IF
		
	EN_RobotMessaging.autoCycleFinished:	//	Re start auto sequencer
		diActualSeqStep						:=	EN_RobotMessaging.autoStarts;
END_CASE
END_METHOD

METHOD Init
//	Keep sequencer in range
	IF (diActualSeqStep<0) OR  (diActualSeqStep>999) THEN
		diActualSeqStep						:=	0;
	END_IF

CASE diActualSeqStep OF
	EN_RobotMessaging.initStart:			//	Wait for init start  perrmissive
		RobotIO.diout_SequenceCmd			:=	EN_RobotMessaging.clearedCmd;
		RobotIO.bout_MotorsOFF				:=	FALSE;
		RobotIO.bout_MotorsON				:=	FALSE;
		RobotIO.bout_PPToMain				:=	FALSE;
		RobotIO.bout_ResetEStop				:=	FALSE;
		RobotIO.bout_Start					:=	FALSE;
		bInit_Finished						:=	FALSE;
		ton_pulse.IN						:= 	FALSE;
		
		IF bInit_StartPermissive THEN
			RobotIO.bout_Stop				:=	(RobotIO.bin_MainTaskExecuting) AND (NOT RobotIO.bin_SystemInputBusy) AND (NOT ton_StepTimeout.Q);
	
			tmStepTimeout					:=	T#1S;
			ton_StepTimeout.IN				:=	RobotIO.bout_Stop OR RobotIO.bin_SystemInputBusy;
			
			IF NOT RobotIO.bin_MainTaskExecuting THEN
				diActualSeqStep				:=	EN_RobotMessaging.turnMotorsOFF;
			END_IF
		
		ELSE
			ton_StepTimeout.IN				:= FALSE;
		END_IF
		
	EN_RobotMessaging.turnMotorsOFF:		//	Turn OFF Motors
		RobotIO.bout_MotorsON				:=	FALSE;
		RobotIO.bout_MotorsOFF				:=	(RobotIO.bin_MotorsON OR (NOT robotio.bin_MotorsOFF)) AND (NOT RobotIO.bin_SystemInputBusy) AND (NOT ton_StepTimeout.Q);
		
		tmStepTimeout						:=	T#1S;
		ton_StepTimeout.IN					:=	RobotIO.bout_MotorsOFF OR RobotIO.bin_SystemInputBusy;
		
		IF ((NOT RobotIO.bin_MotorsON) AND robotio.bin_MotorsOFF) THEN
			diActualSeqStep					:=	EN_RobotMessaging.waitRobotInAuto;
		END_IF
		
	EN_RobotMessaging.waitRobotInAuto:		//	Wait robot is in auto
		tmStepTimeout						:=	T#1S;
		ton_StepTimeout.IN					:=	(NOT RobotIO.bin_AutoON) OR RobotIO.bin_SystemInputBusy;
		
		IF ( RobotIO.bin_AutoON) THEN
			diActualSeqStep					:=	EN_RobotMessaging.resetEStop;
		END_IF
			
	EN_RobotMessaging.resetEStop:			//	Reset E Stop
		RobotIO.bout_ResetEStop				:=	RobotIO.bin_EStop AND (NOT RobotIO.bin_SystemInputBusy) AND (NOT ton_StepTimeout.Q);
		
		tmStepTimeout						:=	T#1S;
		ton_StepTimeout.IN					:=	RobotIO.bout_ResetEStop OR RobotIO.bin_SystemInputBusy;
		
		IF (NOT RobotIO.bin_EStop) THEN
			diActualSeqStep					:=	EN_RobotMessaging.PPToMain;
		END_IF
		
	EN_RobotMessaging.PPToMain:				//	PP to Main
		ton_pulse.IN						:=	(NOT RobotIO.bin_PPMoved) AND (NOT RobotIO.bin_SystemInputBusy) AND (NOT ton_StepTimeout.Q);
		RobotIO.bout_PPToMain				:=	(NOT ton_pulse.Q) AND (ton_pulse.ET>T#0S) AND (ton_pulse.ET<ton_pulse.PT);
		
		tmStepTimeout						:=	T#1S;
		ton_StepTimeout.IN					:=	RobotIO.bout_PPToMain OR RobotIO.bin_SystemInputBusy;
		
		IF RobotIO.bin_PPMoved THEN
			diActualSeqStep					:=	EN_RobotMessaging.turnMotorsON;
		END_IF
		
	EN_RobotMessaging.turnMotorsON:			//	Motors ON
		ton_pulse.IN						:=	((NOT RobotIO.bin_MotorsON) OR RobotIO.bin_MotorsOFF) AND (NOT RobotIO.bin_SystemInputBusy) AND (NOT ton_StepTimeout.Q);
		RobotIO.bout_MotorsON				:=	(NOT ton_pulse.Q) AND (ton_pulse.ET>T#0S) AND (ton_pulse.ET<ton_pulse.PT);
		
		tmStepTimeout						:=	T#1S;
		ton_StepTimeout.IN					:=	RobotIO.bout_MotorsON OR RobotIO.bin_SystemInputBusy;
		
		IF (RobotIO.bin_MotorsON AND (NOT RobotIO.bin_MotorsOFF)) THEN
			diActualSeqStep					:=	EN_RobotMessaging.startTaskExecuion;
		END_IF
		
	EN_RobotMessaging.startTaskExecuion:	//	Start Main Task
		RobotIO.bout_Start					:=	(NOT RobotIO.bin_MainTaskExecuting) AND (NOT RobotIO.bin_SystemInputBusy) AND (NOT ton_StepTimeout.Q);
		
		tmStepTimeout						:=	T#1S;
		ton_StepTimeout.IN					:=	RobotIO.bout_Start OR RobotIO.bin_SystemInputBusy;
		
		IF RobotIO.bin_MainTaskExecuting THEN
			diActualSeqStep					:=	EN_RobotMessaging.waitInitFinihsed;
		END_IF
		
	EN_RobotMessaging.waitInitFinihsed:		//	Wait init finished or ask for permissive to execute retrieval because of robot manually jogged
		tmStepTimeout						:=	T#1S;
		ton_StepTimeout.IN					:=	TRUE;
		
		IF (RobotIO.diin_Sequencer=EN_RobotMessaging.initFinished) OR (RobotIO.diin_Sequencer=EN_RobotMessaging.waitRetrievalPerm) THEN
			diActualSeqStep					:=	RobotIO.diin_Sequencer;
		END_IF
		
	EN_RobotMessaging.waitRetrievalPerm:	//	Wait retrieval permissive from HMI and Handle Hand Shake with robot
		tmStepTimeout						:=	T#5S;
		ton_StepTimeout.IN					:=	TRUE;
		
		IF (RobotIO.diin_Sequencer=EN_RobotMessaging.waitRetrievalPerm) AND bRetrievalPermissive THEN
			RobotIO.diout_SequenceCmd		:=	EN_RobotMessaging.ok;
		ELSE
			RobotIO.diout_SequenceCmd		:=	EN_RobotMessaging.clearedCmd;
			diActualSeqStep					:=	EN_RobotMessaging.waitInitFinihsed;
		END_IF
		
	EN_RobotMessaging.stopTaskExecution:	//	Stop program execution
		RobotIO.bout_Stop					:=	RobotIO.bin_MainTaskExecuting AND (NOT RobotIO.bin_SystemInputBusy) AND (NOT ton_StepTimeout.Q);
		
		tmStepTimeout						:=	T#1S;
		ton_StepTimeout.IN					:=	RobotIO.bout_Stop OR RobotIO.bin_SystemInputBusy;
		
		IF (NOT RobotIO.bin_MainTaskExecuting) THEN
			diActualSeqStep					:=	EN_RobotMessaging.initEndMotorsOFF;
		END_IF
		
	EN_RobotMessaging.initEndMotorsOFF:		// Turn Motors OFF
		RobotIO.bout_MotorsOFF				:=	(RobotIO.bin_MotorsON OR (NOT RobotIO.bin_MotorsOFF)) AND (NOT RobotIO.bin_SystemInputBusy) AND (NOT ton_StepTimeout.Q);
		
		tmStepTimeout						:=	T#1S;
		ton_StepTimeout.IN					:=	RobotIO.bout_MotorsOFF OR RobotIO.bin_SystemInputBusy;
		
		IF (NOT RobotIO.bin_MotorsON) AND RobotIO.bin_MotorsOFF THEN
			diActualSeqStep					:=	EN_RobotMessaging.initFinished;
		END_IF
		
	EN_RobotMessaging.initFinished:			//	Init Finished
		bInit_Finished						:=	TRUE;
END_CASE
END_METHOD

METHOD IO
VAR
	pDint									: POINTER TO DINT;
	pReal									: POINTER TO REAL;
END_VAR
//	Processing protocol raw INPUT data : BITS
	RobotIO.bin_EStop 						:= RobotIO.eipInputs.byteArray[0].0;
	RobotIO.bin_PPMoved 					:= RobotIO.eipInputs.byteArray[0].1;
	RobotIO.bin_MotorsOFF 					:= RobotIO.eipInputs.byteArray[0].2;
	RobotIO.bin_MotorsON					:= RobotIO.eipInputs.byteArray[0].3;
	RobotIO.bin_SystemInputBusy				:= RobotIO.eipInputs.byteArray[0].4;
	RobotIO.bin_RunchainOK 					:= RobotIO.eipInputs.byteArray[0].5;
	RobotIO.bin_AutoON 						:= RobotIO.eipInputs.byteArray[0].6;
	RobotIO.bin_MainTaskExecuting 			:= RobotIO.eipInputs.byteArray[0].7;
	RobotIO.bin_SMBBatery 					:= RobotIO.eipInputs.byteArray[1].0;
	RobotIO.bin_RobotNotMoving				:= RobotIO.eipInputs.byteArray[1].1;
	
	bSafetyBoxPick_OutOfZone 				:= RobotIO.eipInputs.byteArray[1].2;
	bSafetyBoxPlace_OutOfZone 				:= RobotIO.eipInputs.byteArray[1].3;
	bSafetyBoxReject_OutOfZone 				:= RobotIO.eipInputs.byteArray[1].4;
	bPick_AllMaterialPicked					:= RobotIO.eipInputs.byteArray[1].5;
	
	RobotIO.bin_almRetCyl01 				:= RobotIO.eipInputs.byteArray[1].6;
	RobotIO.bin_almExtCyl01					:= RobotIO.eipInputs.byteArray[1].7;
	RobotIO.bin_almBothSnsrCyl01			:= RobotIO.eipInputs.byteArray[2].0;
	RobotIO.bin_almRetCyl02 				:= RobotIO.eipInputs.byteArray[2].1;
	RobotIO.bin_almExtCyl02					:= RobotIO.eipInputs.byteArray[2].2;
	RobotIO.bin_almBothSnsrCyl02			:= RobotIO.eipInputs.byteArray[2].3;
	RobotIO.bin_almRetCyl03 				:= RobotIO.eipInputs.byteArray[2].4;
	RobotIO.bin_almExtCyl03					:= RobotIO.eipInputs.byteArray[2].5;
	RobotIO.bin_almBothSnsrCyl02			:= RobotIO.eipInputs.byteArray[2].6;
	
//	Processing protocol raw INPUT data : BYTES
	pDint 									:= ADR(RobotIO.eipInputs.byteArray[8]);
	RobotIO.diin_Sequencer					:= pDint^;
	
//	Processing protocol raw OUTPUT data : BITS
	RobotIO.eipOutputs.byteArray[0].0 		:= RobotIO.bout_ResetEStop;
	RobotIO.eipOutputs.byteArray[0].1 		:= RobotIO.bout_PPToMain;
	RobotIO.eipOutputs.byteArray[0].2 		:= RobotIO.bout_MotorsOFF;
	RobotIO.eipOutputs.byteArray[0].3 		:= RobotIO.bout_MotorsON;
	RobotIO.eipOutputs.byteArray[0].4 		:= RobotIO.bout_Stop;
	RobotIO.eipOutputs.byteArray[0].5 		:= RobotIO.bout_Start;
	
// In initializaion safety box is bypassed for robot can retrieval
	IF diActualSeqStep=EN_RobotMessaging.waitInitFinihsed OR diActualSeqStep=EN_RobotMessaging.waitRetrievalPerm THEN
		RobotIO.eipOutputs.byteArray[0].6 	:= TRUE;
		RobotIO.eipOutputs.byteArray[0].7 	:= TRUE;
		RobotIO.eipOutputs.byteArray[1].0 	:= TRUE;
	ELSE
		RobotIO.eipOutputs.byteArray[0].6 	:= bSafetyBoxPick_Permissive;
		RobotIO.eipOutputs.byteArray[0].7 	:= bSafetyBoxPlace_Permissive;
		RobotIO.eipOutputs.byteArray[1].0 	:= bSafetyBoxReject_Permissive;
	END_IF
	
// 8 bits array for positions in reject cart
	RobotIO.eipOutputs.byteArray[1].1		:= bReject_MaterialRequest[0];
	RobotIO.eipOutputs.byteArray[1].2		:= bReject_MaterialRequest[1];
	RobotIO.eipOutputs.byteArray[1].3		:= bReject_MaterialRequest[2];
	RobotIO.eipOutputs.byteArray[1].4		:= bReject_MaterialRequest[3];
	RobotIO.eipOutputs.byteArray[1].5		:= bReject_MaterialRequest[4];
	RobotIO.eipOutputs.byteArray[1].6		:= bReject_MaterialRequest[5];
	RobotIO.eipOutputs.byteArray[1].7		:= bReject_MaterialRequest[6];
	RobotIO.eipOutputs.byteArray[2].0		:= bReject_MaterialRequest[7];
	
//	Dry cycle activation bit
	RobotIO.eipOutputs.byteArray[2].1		:= bDryCycleON;
	
// Processing protocol raw OUTPUT data : BYTES
	pDint 									:= ADR(RobotIO.eipOutputs.byteArray[8]);
	pdint^									:= RobotIO.diout_SequenceCmd;
	pReal 									:= ADR(RobotIO.eipOutputs.byteArray[12]);
	pReal^									:= RobotIO.rout_XCompensation;
	pReal 									:= ADR(RobotIO.eipOutputs.byteArray[16]);
	pReal^									:= RobotIO.rout_ZCompensation;
END_METHOD

METHOD Manual
VAR
	manualCommand				:	EN_RobotMessaging;
END_VAR
IF (RobotIO.diin_Sequencer=EN_RobotMessaging.clearedCmd) THEN 
	RobotIO.diout_SequenceCmd			:=	manualCommand;
ELSE
	RobotIO.diout_SequenceCmd			:=	EN_RobotMessaging.clearedCmd;
END_IF
END_METHOD

METHOD Pause
RobotIO.bout_Stop						:=	RobotIO.bin_MainTaskExecuting AND (NOT ton_StepTimeout.Q);
RobotIO.bout_MotorsOFF					:=	NOT RobotIO.bin_MainTaskExecuting AND RobotIO.bin_RobotNotMoving AND RobotIO.bin_MotorsON;
ton_StepTimeout.IN						:=	RobotIO.bout_Stop;
ton_pulse.IN							:=	FALSE;
END_METHOD

METHOD Stop
Pause();
bInit_Finished 							:=	FALSE;
diActualSeqStep							:=	0;
END_METHOD

END_FUNCTION_BLOCK

// ---- POUs/01-DevicesFB/Scanner/FB_Scanner.TcPOU
FUNCTION_BLOCK FB_Scanner EXTENDS FB_Device

//Alarms:
//	 1:= No conectado
//   2:= Deshabilitado
//   3:= Error de lectura
//   4:= Error en cambio de programa
//   5:= Timeout

VAR_INPUT
	bIn_Trigger						: BOOL;
	bIn_Reset						: BOOL;
	bDisable						: BOOL;
	iTotalRetries					: USINT		:= 2;
	
	//Time before alarm set
	Timeout							: TIME;
END_VAR

VAR_OUTPUT
	//String code
		sCode						: STRING;
		bCompleted					: BOOL;
		bConnected					: BOOL;
END_VAR
VAR
	tmrAlarm						: TON;
	r_trig							: R_TRIG;
	iStep							: USINT	:= 0;
	
	//To scanner
	bOutReadRequest 		AT%Q*	: BOOL;
	bOutErrorClear 			AT%Q*	: BOOL;
	bOutReadClear 			AT%Q*	: BOOL;
	
	//From scanner
	bInReadFailure			AT%I*	: BOOL;
	bInBusy					AT%I*	: BOOL;
	bInReady				AT%I*	: BOOL;
	bInReadComplete			AT%I*	: BOOL;
	iCommStatus 			AT%I*	: UINT;
		
		//Check the array lenght (this is 127 array, from keyence sr2000)
	ResultData				AT%I*	: ARRAY[0..127]OF BYTE;
	iResultDataSize			AT%I* 	: UINT;
	
	iRetryCounter				:USINT;
	
END_VAR

//If it's disabled, send the alarm and set on the code
IF bDisable THEN
	bCompleted:= TRUE;
	sCode:= 'Disabled';
	sAlarm:= 'Disabled';//Deshabilitado
	RETURN;	
END_IF

//Update communication status
bConnected:= iCommStatus = 0;

CASE iStep OF
	
	0:		//Wait for trigger
	
		IF bIn_Trigger THEN
			iRetryCounter:= 0;
			iStep:= iStep+1;	
		END_IF
		
	1:		//Check scanner disabled
	
		IF bDisable THEN
			sAlarm:= 'Disabled';//Scanner disabled
			sCode:= 'Disabled';
			iStep:= 9;
		END_IF
		
		iStep:= iStep+1;		

	2:		//Check connection
	
		IF bConnected THEN
			iStep:= iStep+1;
		ELSE
			sAlarm:= 'Disconnected';//Not connection
			iStep:= 1;
		END_IF

	
	3:		//Variable reset
	
		Reset();	
		iStep:= iStep+1;
	
	4:		//Request to read code
	
		bOutReadRequest:= TRUE;
		iStep:= iStep+1;
	
	5:		//Confirm read request
		
		IF bInBusy THEN
			bOutReadRequest:= FALSE;		
			iStep:= iStep+1;			
		END_IF
	
	6:		//Wait for read completion
	
		tmrAlarm(IN:= TRUE, PT:= Timeout);
		
		IF bInReadComplete THEN		
			iStep:= iStep+1;
		ELSIF tmrAlarm.Q THEN
			sAlarm:='Code read timeout';//Code read timeout
			iStep:= 7;
		END_IF
	
	7:		//Check for scan failure
	
		IF bInReadFailure THEN
			IF  iRetryCounter< iTotalRetries THEN
				iRetryCounter:= iRetryCounter+1;
				iStep:= 1;
				RETURN;				
 			END_IF  									
			sAlarm:= 'Read code error';//Error de lectura de codigo
				
		END_IF
		iStep:= iStep+1;

	8:		//Read data
	
		//Move the byte data to the string result code
		MEMMOVE(
			destAddr	:= ADR(sCode),
			srcAddr		:= ADR(ResultData),
			n			:= iResultDataSize);							
			iStep:= iStep+1;
	
	9:		//Wait for trigger remove
	
		bCompleted:= TRUE;
		IF NOT bIn_Trigger THEN
			iStep:= 0;
		END_IF
	
END_CASE

ACTION Reset:
tmrAlarm(IN:= FALSE);
sCode := '';  
sAlarm := '';
bOutReadRequest := FALSE;
bInReadComplete := FALSE;
bOutReadClear := TRUE;
bCompleted := FALSE;
END_ACTION

END_FUNCTION_BLOCK

// ---- POUs/01-DevicesFB/TrayFeeder/FB_TrayFeeder.TcPOU
FUNCTION_BLOCK FB_TrayFeeder EXTENDS FB_Machine
VAR_INPUT
	// Material tray move permissive
	bSafetyBoxDeliver_permissive		: BOOL;
	
	// Ask for replace material tray
	bChangeTrayRequest 					: BOOL;
END_VAR
VAR_OUTPUT
	// Material tray zone is safe to enter in
	bSafetyBoxDeliver_isSafe			: BOOL;
	
	// Good material is on work position
	bMaterial_ReadyToPick				: BOOL;
END_VAR
VAR
	// Input: HMI Piece is good for process
	bScanningPieceIsOK					: BOOL;
	// Input: HMI Piece is no good for process
	bScanningPieceIsNG					: BOOL;
	
	// Structure for IO Mapping
	TrayFeederIO						: ST_TrayFeederIO;
END_VAR

super^.MachineMain();

METHOD Alarm
VAR
	// R Trigger VAr
	rTrigger							: R_TRIG;
	// Step in wich timeout occur
	diTimeoutStep						: DINT;
	// Actual Timed Out Sequence Step Code
	sSequenceCode						: STRING;
	
	// Async Process Concatenated Alarm Codes
	sAsyncAlarmCodes					: STRING;
END_VAR
// 	Timeout preset valuie setting
	IF ton_StepTimeout.PT<>tmStepTimeout THEN
		ton_StepTimeout.PT					:= tmStepTimeout;
	END_IF

// 	TON for step timeout
	ton_StepTimeout(IN:=((NOT ton_StepTimeout.Q) AND (diLastActiveStep=diActualSeqStep)));

// 	Following of sequence for setting timeout
	IF diLastActiveStep<>diActualSeqStep THEN
		diLastActiveStep					:= diActualSeqStep;
	END_IF

// 	For setting acual timed out step alarm code
	rTrigger(CLK:=ton_StepTimeout.Q);
	IF rTrigger.Q THEN
		diTimeoutStep := diActualSeqStep;
		CASE diTimeoutStep OF
		// Init process timeouts
			EN_RobotMessaging.initStart: 			sSequenceCode := '';
			
		// Robot Auto
			EN_RobotMessaging.autoStarts:			sSequenceCode := '';
			
		END_CASE
		sSequenceCode:= CONCAT(STR1:=sSequenceCode,STR2:=sDeviceID);
		sSequenceCode:= CONCAT(STR1:=sSequenceCode,STR2:=',');
	END_IF

// 	For deleting last sequence alarm code automatically
	IF (diActualSeqStep<>diTimeoutStep AND diTimeoutStep<>EN_RobotMessaging.clearedCmd)THEN
		sSequenceCode:= '';
		diTimeoutStep:= EN_RobotMessaging.clearedCmd;
	END_IF

// 	For setting no lineal processes alarms
	// Tray Feeder is not in auto mode
	sAsyncAlarmCodes:= AlarmCodesHandling(sConcatCodes:=sAsyncAlarmCodes,sCode:='WFEEDOMD01',sIDToAdd:=sDeviceID,bActive:=NOT(TrayFeederIO.diin_StationStatus=EN_StationStatus.maintenance));
	// Tray Feeder connection failed
	sAsyncAlarmCodes:= AlarmCodesHandling(sConcatCodes:=sAsyncAlarmCodes,sCode:='EFEEDCON01',sIDToAdd:=sDeviceID,bActive:=(TrayFeederIO.uiin_ConnectionStatus=0));
	// Tray Feeder EStop pressed
	sAsyncAlarmCodes:= AlarmCodesHandling(sConcatCodes:=sAsyncAlarmCodes,sCode:='SFEEDALA01',sIDToAdd:=sDeviceID,bActive:=(TrayFeederIO.diin_StationStatus=EN_StationStatus.estopped));
	// Tray Feeder Stucked in place safe box
	sAsyncAlarmCodes:= AlarmCodesHandling(sConcatCodes:=sAsyncAlarmCodes,sCode:='EFEEDSTU01',sIDToAdd:=sDeviceID,bActive:=((NOT TrayFeederIO.bin_SafetyBoxPlace_OutOfZone) AND (TrayFeederIO.bout_SafetyBoxPlace_Permissive)));
	// Safety gratings interrupted impede machine operation
	sAsyncAlarmCodes:= AlarmCodesHandling(sConcatCodes:=sAsyncAlarmCodes,sCode:='WFEEDSTU01',sIDToAdd:=sDeviceID,bActive:=(FALSE));
	
// 	Concat all alarm codes
	sAlarm:= CONCAT(STR1:=sSequenceCode,STR2:=sAsyncAlarmCodes);
END_METHOD

METHOD Auto_Feeder
//	 Keep sequencer in range
	IF (diActualSeqStep<1000) OR (diActualSeqStep>1999) THEN
		diActualSeqStep												:=1000;
	END_IF

CASE diActualSeqStep OF
	EN_TrayFeederMessaging.autoStart:
		IF NOT ST_TrayFeederIO.bin_AutoOn THEN
			ST_TrayFeederIO.bout_Start 								:=TRUE;
		END_IF
		IF ST_TrayFeederIO.bin_AutoOn THEN
			ST_TrayFeederIO.bout_Start								:=FALSE;
			diActualSeqStep											:= EN_TrayFeederMessaging.readyToPick;
		END_IF
	EN_TrayFeederMessaging.readyToPick:
		IF ST_TrayFeederIO.bout_readyToPick AND ST_TrayFeederIO.bin_SafetyBoxPlace_OutOfZone THEN
			ST_TrayFeederIO.bout_SafetyBoxPlace_Permissive			:=TRUE;
			diActualSeqStep											:=En_TrayFeederMessaging.picking;
		END_IF
	En_TrayFeederMessaging.picking:
		IF NOT ST_TrayfeederIO.bin_SafetyBoxPlace_OutOfZone THEN
			ST_TrayFeederIO.bout_SafetyBoxPlace_Permissive			:=FALSE;
			diActualSeqStep											:=En_TrayFeederMessaging.picking;
		END_IF
END_CASE
END_METHOD

METHOD Auto_Gantry
//	 Keep sequencer in range
	IF (diActualSeqStep<1000) OR (diActualSeqStep>1999) THEN
		diActualSeqStep							:=	1000;
	END_IF

CASE	diActualSeqStep OF
	EN_TrayFeederMessaging.autoStart:	//	Get down empty lifter to traslation height
	//	Check if have tray on lifter
	//	Move empty lifter to feed tray tower position
	//	Lift feed tray tower to unlock height
	//	Release feed tray tower
	//	Get down feed tray tower to re lock height
	//	Re lock feed tray tower
	//	Get down new tray to traslation height
	//	Move new tray to work position
	//	Lift new tray to work position
	//	Wait tray change request
		bMaterial_ReadyToPick					:=	TrayFeederIO.bin_delivery_trayReady;
	//	Move to tray reject position
	//	Lift reject tray tower to unlock height
	//	Unlock reject tray tower
	//	Lift reject tray tower to re lock height
	//	Re lock reject tray tower
	//	Reset Auto Sequencer
END_CASE
END_METHOD

METHOD Init
//	 Keep sequencer in range
	IF (diActualSeqStep<0) OR (diActualSeqStep>999) THEN
		diActualSeqStep							:=	0;
	END_IF

CASE diActualSeqStep OF
	EN_TrayFeederMessaging.waitInitStart:				//	When init start bit permissive, set init start output and wait feeder confirm init started
		IF NOT ST_TrayFeederIO.bin_initFinished AND ST_TrayFeederIO.bin_SafetyBoxPlace_OutOfZone THEN
			TrayFeederIO.bout_Reset	:=	TRUE;
		END_IF
		IF ST_TrayFeederIO.bin_initFinished THEN
			diActualSeqStep							:=999;
		END_IF
END_CASE
END_METHOD

METHOD IO
VAR
	pDint										: POINTER TO DINT;
END_VAR
// 	FB Direct Inputs
	TrayFeederIO.bout_SafetyBoxPlace_Permissive		:= bSafetyBoxDeliver_permissive;
	TrayFeederIO.bout_delivery_trayChangeRequest	:= bChangeTrayRequest;
	TrayFeederIO.bout_readyToScan					:= bPart_ReadyToScan;
	TrayFeederIO.bout_readyToPick					:= bMaterial_ReadyToPick;
	
	TrayFeederIO.bout_scannninPieceIsOK				:= bScanningPieceIsOK;
	TrayFeederIO.bout_scannninPieceIsNG				:= bScanningPieceIsNG;
	
//	Processing protocol raw data : INPUT BITS
	TrayFeederIO.bin_ServosFailure					:= TrayFeederIO.eipInputs.byteArray[0].0;
	TrayFeederIO.bin_initFinished					:= TrayFeederIO.eipInputs.byteArray[0].1;
	TrayFeederIO.bin_SafetyBoxPlace_OutOfZone		:= TrayFeederIO.eipInputs.byteArray[0].2;
	TrayFeederIO.bin_inScanningPosition				:= TrayFeederIO.eipInputs.byteArray[0].3;
	TrayFeederIO.bin_delivery_trayReady				:= TrayFeederIO.eipInputs.byteArray[0].4;
	
//	Processing protocol raw data : INPUT BYTES
	pDint											:= ADR(TrayFeederIO.eipInputs.byteArray[8]);
	TrayFeederIO.diin_StationStatus					:= pDint^;
	pDint 											:= ADR(TrayFeederIO.eipInputs.byteArray[12]);
	TrayFeederIO.diin_Sequencer						:= pDint^;
	
//	Processing protocol raw data : OUTPUT BITS
	TrayFeederIO.eipOutputs.byteArray[0].0 	:= TrayFeederIO.bout_Reset;
	TrayFeederIO.eipOutputs.byteArray[0].1	:= TrayFeederIO.bout_Start;
	TrayFeederIO.eipOutputs.byteArray[0].2	:= TrayFeederIO.bout_Stop;
	TrayFeederIO.eipOutputs.byteArray[0].3	:= TrayFeederIO.bout_Init_startPermissive;
	TrayFeederIO.eipOutputs.byteArray[0].4	:= TrayFeederIO.bout_SafetyBoxPlace_Permissive;
	TrayFeederIO.eipOutputs.byteArray[0].5	:= TrayFeederIO.bout_scannninPieceIsOK;
	TrayFeederIO.eipOutputs.byteArray[0].6	:= TrayFeederIO.bout_scannninPieceIsNG;
	TrayFeederIO.eipOutputs.byteArray[0].7	:= TrayFeederIO.bout_delivery_trayChangeRequest;
	
// 	Processing protocol raw data : OUTPUT BYTES
	pDint 											:= ADR(TrayFeederIO.eipOutputs.byteArray[8]);
	pdint^											:= TrayFeederIO.diout_SequenceCmd;
	
// 	FB Direct Outputs
	bSafetyBoxDeliver_isSafe						:= TrayFeederIO.bin_SafetyBoxPlace_OutOfZone;
END_METHOD

METHOD Manual
//	Keep sequencer in range
	IF (diActualSeqStep<2000) OR (diActualSeqStep>2999) THEN
		diActualSeqStep							:=	0;
	END_IF
END_METHOD

METHOD Pause
TrayFeederIO.bout_Stop						:=(TrayFeederIO.diin_StationStatus=EN_StationStatus.running);
END_METHOD

{warning 'Add method implementation '}
METHOD Stop
END_METHOD

END_FUNCTION_BLOCK

// ---- POUs/01-DevicesFB/Vaccum/FB_Vacuum.TcPOU
FUNCTION_BLOCK FB_Vacuum EXTENDS FB_Device
VAR_INPUT
	bGrip							: BOOL;
	Timeout							: TIME;
END_VAR
VAR_OUTPUT
	Vacuum_Ok						: BOOL;
	Blow_Ok							: BOOL;
END_VAR
VAR
	VacuumValve				AT %Q*	: BOOL;
	BlowValve				AT %Q*	: BOOL;
	VaccumSensor			AT %I*	: BOOL;
	tmrBlow							: TP;
END_VAR

//	If execute grip input then grip
	VacuumValve						:=	bGrip;
	BlowValve						:=	(NOT bGrip) AND VaccumSensor;

//	Assing valiue to function block status
	Vacuum_Ok							:= VaccumSensor AND NOT BlowValve;
	Blow_Ok								:= BlowValve AND NOT VacuumValve;

//	For setting alarms
	Alarm();

METHOD Alarm
//	Timer for set action executing timeout alarm
	ton_StepTimeout(		IN:=(VacuumValve AND (NOT VaccumSensor)) OR (BlowValve AND VaccumSensor),
							PT:=Timeout);

//	For no vacc sensor feedback alarm setting
	AlarmCodesHandling(sConcatCodes:=sAlarm,sCode:='EVACUDET01 ',sIDToAdd:=sDeviceID,bActive:=(VacuumValve AND ton_StepTimeout.Q));
//	For no release success alarm setting
	AlarmCodesHandling(sConcatCodes:=sAlarm,sCode:='EVACUDET02 ',sIDToAdd:=sDeviceID,bActive:=(BlowValve AND ton_StepTimeout.Q));
END_METHOD

METHOD Pick : bool
VAR_INPUT	
END_VAR
BlowValve:= FALSE;
VacuumValve:= TRUE;

//IF NOT VaccumSensor THEN
//	SetAlarm('Vacuum not reached!');
//ELSE
//	SetAlarm('');	
//END_IF

Pick := VaccumSensor;
END_METHOD

METHOD Release : bool
VAR_INPUT
	Blow			: BOOL 	:= FALSE;
	BlowPulse		: TIME	:= T#100MS;
END_VAR
VacuumValve:= FALSE;
tmrBlow(In:= TRUE, PT:= BlowPulse);

IF blow AND tmrBlow.Q THEN
	BlowValve:= TRUE;
ELSE
	BlowValve:= FALSE;		
END_IF



Release := NOT VaccumSensor AND tmrBlow.Q;
END_METHOD

END_FUNCTION_BLOCK
